C05505=1108.942,119.637,-59.989,-179.645,8.357,149.505
C05506=1108.947,119.424,-59.972,-179.646,8.354,149.505
C05507=1108.951,119.210,-59.955,-179.648,8.352,149.505
C05508=1108.955,118.996,-59.937,-179.649,8.349,149.504
C05509=1108.959,118.783,-59.919,-179.651,8.345,149.504
C05510=1108.963,118.569,-59.902,-179.652,8.342,149.504
C05511=1108.967,118.356,-59.885,-179.653,8.340,149.504
C05512=1108.971,118.142,-59.867,-179.655,8.337,149.503
C05513=1108.975,117.929,-59.849,-179.656,8.334,149.503
C05514=1108.979,117.680,-59.829,-179.658,8.331,149.503
C05515=1108.985,117.430,-59.809,-179.660,8.327,149.503
C05516=1108.989,117.181,-59.788,-179.661,8.324,149.502
C05517=1108.994,116.932,-59.768,-179.664,8.321,149.502
C05518=1108.998,116.683,-59.748,-179.666,8.317,149.502
C05519=1109.004,116.433,-59.727,-179.667,8.313,149.501
C05520=1109.008,116.184,-59.707,-179.669,8.310,149.501
C05521=1109.013,115.935,-59.687,-179.671,8.307,149.501
C05522=1109.017,115.686,-59.666,-179.672,8.303,149.500
C05523=1109.023,115.436,-59.646,-179.674,8.300,149.500
C05524=1109.027,115.187,-59.626,-179.676,8.297,149.500
C05525=1109.031,114.938,-59.605,-179.677,8.293,149.499
C05526=1109.036,114.689,-59.586,-179.679,8.290,149.499
C05527=1109.041,114.441,-59.566,-179.681,8.287,149.499
C05528=1109.046,114.191,-59.545,-179.683,8.283,149.499
C05529=1109.051,113.942,-59.525,-179.685,8.279,149.498
C05530=1109.056,113.693,-59.505,-179.686,8.277,149.498
C05531=1109.060,113.444,-59.484,-179.688,8.273,149.498
C05532=1109.065,113.194,-59.464,-179.690,8.269,149.497
C05533=1109.069,112.945,-59.444,-179.692,8.266,149.497
C05534=1109.074,112.696,-59.423,-179.693,8.263,149.497
C05535=1109.080,112.447,-59.404,-179.695,8.259,149.497
C05536=1109.084,112.198,-59.383,-179.697,8.256,149.496
C05537=1109.089,111.949,-59.364,-179.698,8.253,149.496
C05538=1109.093,111.700,-59.343,-179.700,8.249,149.496
C05539=1109.098,111.450,-59.324,-179.702,8.246,149.495
C05540=1109.102,111.201,-59.303,-179.704,8.242,149.495
C05541=1109.108,110.952,-59.284,-179.706,8.238,149.495
C05542=1109.112,110.703,-59.264,-179.708,8.235,149.495
C05543=1109.117,110.454,-59.244,-179.709,8.231,149.494
C05544=1109.122,110.205,-59.223,-179.711,8.227,149.494
C05545=1109.127,109.955,-59.203,-179.713,8.224,149.494
C05546=1109.131,109.706,-59.183,-179.715,8.220,149.493
C05547=1109.137,109.457,-59.164,-179.717,8.216,149.493
C05548=1109.141,109.208,-59.143,-179.719,8.213,149.493
C05549=1109.146,108.959,-59.124,-179.721,8.209,149.493
C05550=1109.150,108.710,-59.103,-179.723,8.206,149.492
C05551=1109.156,108.461,-59.084,-179.725,8.202,149.492
C05552=1109.160,108.211,-59.064,-179.726,8.198,149.491
C05553=1109.165,107.962,-59.044,-179.729,8.195,149.491
C05554=1109.170,107.713,-59.024,-179.731,8.191,149.491
C05555=1109.174,107.463,-59.005,-179.732,8.187,149.491
C05556=1109.179,107.215,-58.985,-179.734,8.185,149.490
C05557=1109.184,106.965,-58.965,-179.735,8.181,149.490
C05558=1109.188,106.716,-58.946,-179.737,8.177,149.490
C05559=1109.193,106.467,-58.926,-179.739,8.173,149.489
C05560=1109.198,106.218,-58.906,-179.741,8.170,149.489
C05561=1109.203,105.969,-58.887,-179.743,8.166,149.489
C05562=1109.207,105.755,-58.869,-179.745,8.162,149.488
C05563=1109.210,105.542,-58.853,-179.746,8.159,149.488
C05564=1109.215,105.328,-58.835,-179.748,8.156,149.488
C05565=1109.219,105.114,-58.819,-179.749,8.153,149.488
C05566=1109.223,104.901,-58.802,-179.750,8.150,149.487
C05567=1109.227,104.687,-58.785,-179.752,8.146,149.487
C05568=1109.231,104.473,-58.768,-179.754,8.144,149.487
C05569=1109.235,104.259,-58.752,-179.755,8.141,149.486
C05570=1109.240,104.010,-58.732,-179.757,8.137,149.486
C05571=1109.245,103.761,-58.713,-179.758,8.133,149.486
C05572=1109.249,103.512,-58.692,-179.760,8.129,149.485
C05573=1109.255,103.263,-58.673,-179.762,8.126,149.485
C05574=1109.260,103.013,-58.653,-179.763,8.122,149.484
C05575=1109.264,102.764,-58.634,-179.765,8.118,149.484
C05576=1109.269,102.515,-58.615,-179.767,8.114,149.484
C05577=1109.274,102.266,-58.595,-179.769,8.111,149.483
C05578=1109.278,102.016,-58.576,-179.770,8.107,149.483
C05579=1109.284,101.767,-58.556,-179.772,8.103,149.482
C05580=1109.288,101.518,-58.537,-179.774,8.099,149.482
C05581=1109.292,101.269,-58.517,-179.776,8.096,149.482
C05582=1109.297,101.020,-58.498,-179.777,8.092,149.481
C05583=1109.302,100.771,-58.478,-179.778,8.089,149.481
C05584=1109.307,100.522,-58.459,-179.780,8.085,149.481
C05585=1109.312,100.273,-58.440,-179.781,8.081,149.480
C05586=1109.316,100.023,-58.420,-179.783,8.077,149.480
C05587=1109.322,99.774,-58.401,-179.785,8.073,149.479
C05588=1109.326,99.525,-58.382,-179.787,8.069,149.479
C05589=1109.331,99.276,-58.362,-179.788,8.066,149.479
C05590=1109.336,99.026,-58.343,-179.790,8.062,149.478
C05591=1109.340,98.777,-58.324,-179.791,8.058,149.478
C05592=1109.345,98.528,-58.304,-179.792,8.055,149.477
C05593=1109.350,98.278,-58.285,-179.794,8.051,149.477
C05594=1109.356,98.029,-58.266,-179.796,8.047,149.476
C05595=1109.360,97.780,-58.247,-179.797,8.043,149.476
C05596=1109.365,97.531,-58.228,-179.799,8.039,149.475
C05597=1109.369,97.282,-58.209,-179.800,8.035,149.475
C05598=1109.374,97.032,-58.189,-179.802,8.031,149.475
C05599=1109.379,96.783,-58.170,-179.803,8.028,149.474
C05600=1109.383,96.534,-58.151,-179.805,8.024,149.474
C05601=1109.388,96.285,-58.131,-179.806,8.021,149.473
C05602=1109.393,96.035,-58.113,-179.808,8.017,149.473
C05603=1109.398,95.787,-58.094,-179.809,8.013,149.472
C05604=1109.403,95.537,-58.074,-179.811,8.009,149.472
C05605=1109.407,95.288,-58.055,-179.812,8.006,149.472
C05606=1109.412,95.039,-58.036,-179.814,8.002,149.471
C05607=1109.418,94.789,-58.017,-179.815,7.998,149.471
C05608=1109.422,94.540,-57.998,-179.816,7.994,149.470
C05609=1109.427,94.291,-57.979,-179.818,7.990,149.470
C05610=1109.431,94.042,-57.960,-179.819,7.987,149.469
C05611=1109.437,93.792,-57.941,-179.820,7.983,149.469
C05612=1109.441,93.543,-57.922,-179.822,7.979,149.468
C05613=1109.446,93.294,-57.903,-179.824,7.975,149.468
C05614=1109.450,93.045,-57.884,-179.825,7.971,149.467
C05615=1109.456,92.796,-57.865,-179.826,7.968,149.467
C05616=1109.460,92.546,-57.846,-179.827,7.964,149.466
C05617=1109.465,92.297,-57.827,-179.829,7.960,149.466
C05618=1109.469,92.083,-57.811,-179.830,7.957,149.466
C05619=1109.473,91.870,-57.795,-179.831,7.954,149.465
C05620=1109.478,91.656,-57.778,-179.833,7.950,149.465
C05621=1109.482,91.441,-57.762,-179.833,7.947,149.464
C05622=1109.486,91.228,-57.747,-179.834,7.944,149.464
C05623=1109.490,91.015,-57.730,-179.836,7.941,149.464
C05624=1109.493,90.801,-57.714,-179.837,7.937,149.463
C05625=1109.498,90.587,-57.698,-179.838,7.934,149.463
C05626=1109.503,90.338,-57.678,-179.840,7.930,149.462
C05627=1109.507,90.088,-57.660,-179.841,7.926,149.462
C05628=1109.513,89.840,-57.641,-179.842,7.923,149.461
C05629=1109.517,89.590,-57.623,-179.844,7.919,149.461
C05630=1109.522,89.341,-57.603,-179.844,7.915,149.460
C05631=1109.527,89.091,-57.585,-179.846,7.911,149.460
C05632=1109.531,88.842,-57.566,-179.847,7.907,149.459
C05633=1109.537,88.593,-57.548,-179.849,7.903,149.459
C05634=1109.541,88.344,-57.529,-179.850,7.900,149.458
C05635=1109.547,88.094,-57.510,-179.851,7.896,149.458
C05636=1109.551,87.845,-57.491,-179.852,7.892,149.457
C05637=1109.556,87.596,-57.473,-179.853,7.889,149.457
C05638=1109.561,87.347,-57.454,-179.854,7.884,149.456
C05639=1109.565,87.097,-57.435,-179.856,7.881,149.456
C05640=1109.570,86.848,-57.417,-179.857,7.877,149.455
C05641=1109.576,86.599,-57.398,-179.858,7.873,149.454
C05642=1109.580,86.350,-57.379,-179.860,7.869,149.454
C05643=1109.584,86.100,-57.361,-179.861,7.866,149.454
C05644=1109.590,85.851,-57.343,-179.862,7.862,149.453
C05645=1109.594,85.602,-57.323,-179.863,7.858,149.453
C05646=1109.599,85.353,-57.305,-179.864,7.854,149.452
C05647=1109.604,85.104,-57.286,-179.865,7.851,149.451
C05648=1109.609,84.854,-57.268,-179.867,7.846,149.451
C05649=1109.614,84.605,-57.250,-179.868,7.843,149.450
C05650=1109.619,84.356,-57.231,-179.869,7.839,149.450
C05651=1109.623,84.106,-57.212,-179.870,7.836,149.449
C05652=1109.628,83.857,-57.194,-179.871,7.832,149.449
C05653=1109.633,83.608,-57.176,-179.872,7.828,149.448
C05654=1109.638,83.358,-57.157,-179.873,7.825,149.448
C05655=1109.643,83.109,-57.139,-179.874,7.820,149.447
C05656=1109.647,82.860,-57.120,-179.875,7.817,149.447
C05657=1109.652,82.611,-57.102,-179.877,7.813,149.446
C05658=1109.657,82.361,-57.083,-179.878,7.809,149.446
C05659=1109.662,82.112,-57.065,-179.879,7.805,149.445
C05660=1109.667,81.863,-57.046,-179.880,7.802,149.445
C05661=1109.671,81.613,-57.028,-179.881,7.798,149.444
C05662=1109.676,81.364,-57.010,-179.882,7.794,149.443
C05663=1109.682,81.115,-56.991,-179.883,7.791,149.443
C05664=1109.686,80.866,-56.973,-179.884,7.787,149.442
C05665=1109.691,80.616,-56.954,-179.885,7.783,149.442
C05666=1109.696,80.367,-56.936,-179.887,7.779,149.441
C05667=1109.700,80.118,-56.918,-179.887,7.776,149.441
C05668=1109.706,79.868,-56.900,-179.889,7.772,149.440
C05669=1109.710,79.618,-56.882,-179.889,7.769,149.440
C05670=1109.715,79.370,-56.863,-179.891,7.765,149.439
C05671=1109.720,79.121,-56.845,-179.891,7.761,149.438
C05672=1109.725,78.872,-56.827,-179.892,7.757,149.438
C05673=1109.730,78.622,-56.809,-179.893,7.754,149.437
C05674=1109.734,78.408,-56.793,-179.894,7.751,149.437
C05675=1109.738,78.194,-56.778,-179.895,7.747,149.436
C05676=1109.742,77.980,-56.762,-179.896,7.744,149.436
C05677=1109.747,77.767,-56.746,-179.897,7.741,149.435
C05678=1109.751,77.552,-56.731,-179.898,7.738,149.435
C05679=1109.755,77.339,-56.715,-179.899,7.735,149.435
C05680=1109.759,77.125,-56.699,-179.899,7.731,149.434
C05681=1109.763,76.911,-56.684,-179.900,7.728,149.433
C05682=1109.768,76.662,-56.666,-179.902,7.724,149.433
C05683=1109.773,76.413,-56.647,-179.903,7.720,149.433
C05684=1109.777,76.163,-56.629,-179.904,7.716,149.432
C05685=1109.782,75.914,-56.611,-179.906,7.712,149.432
C05686=1109.787,75.665,-56.593,-179.907,7.708,149.431
C05687=1109.792,75.415,-56.575,-179.909,7.704,149.431
C05688=1109.797,75.166,-56.557,-179.910,7.700,149.430
C05689=1109.802,74.917,-56.539,-179.912,7.696,149.430
C05690=1109.806,74.667,-56.520,-179.913,7.693,149.429
C05691=1109.811,74.418,-56.502,-179.914,7.689,149.428
C05692=1109.816,74.168,-56.485,-179.915,7.685,149.428
C05693=1109.821,73.919,-56.467,-179.917,7.681,149.428
C05694=1109.826,73.670,-56.449,-179.919,7.677,149.427
C05695=1109.831,73.421,-56.431,-179.920,7.673,149.427
C05696=1109.836,73.172,-56.413,-179.921,7.669,149.426
C05697=1109.841,72.922,-56.395,-179.923,7.665,149.426
C05698=1109.845,72.672,-56.377,-179.924,7.661,149.425
C05699=1109.850,72.423,-56.359,-179.926,7.657,149.425
C05700=1109.855,72.174,-56.341,-179.926,7.654,149.424
C05701=1109.860,71.924,-56.324,-179.928,7.649,149.423
C05702=1109.865,71.675,-56.306,-179.929,7.645,149.423
C05703=1109.869,71.426,-56.288,-179.931,7.642,149.423
C05704=1109.874,71.177,-56.270,-179.932,7.637,149.422
C05705=1109.879,70.928,-56.252,-179.933,7.633,149.422
C05706=1109.884,70.679,-56.234,-179.935,7.629,149.421
C05707=1109.889,70.429,-56.217,-179.936,7.625,149.420
C05708=1109.894,70.180,-56.199,-179.938,7.621,149.420
C05709=1109.899,69.931,-56.181,-179.939,7.618,149.420
C05710=1109.904,69.681,-56.163,-179.940,7.614,149.419
C05711=1109.909,69.432,-56.146,-179.941,7.610,149.418
C05712=1109.913,69.182,-56.128,-179.943,7.606,149.418
C05713=1109.918,68.933,-56.110,-179.944,7.602,149.417
C05714=1109.923,68.684,-56.092,-179.946,7.598,149.417
C05715=1109.928,68.434,-56.075,-179.947,7.594,149.417
C05716=1109.933,68.185,-56.057,-179.948,7.590,149.416
C05717=1109.938,67.936,-56.039,-179.950,7.586,149.415
C05718=1109.942,67.686,-56.022,-179.951,7.583,149.415
C05719=1109.947,67.437,-56.004,-179.952,7.578,149.414
C05720=1109.952,67.188,-55.986,-179.953,7.574,149.414
C05721=1109.957,66.938,-55.969,-179.955,7.571,149.414
C05722=1109.962,66.689,-55.951,-179.956,7.566,149.413
C05723=1109.967,66.439,-55.934,-179.958,7.562,149.412
C05724=1109.972,66.190,-55.916,-179.959,7.558,149.412
C05725=1109.977,65.941,-55.899,-179.960,7.555,149.411
C05726=1109.982,65.691,-55.881,-179.961,7.551,149.411
C05727=1109.986,65.442,-55.864,-179.962,7.547,149.410
C05728=1109.991,65.192,-55.847,-179.964,7.543,149.410
C05729=1109.997,64.944,-55.829,-179.966,7.539,149.409
C05730=1110.000,64.730,-55.814,-179.966,7.535,149.409
C05731=1110.005,64.516,-55.799,-179.968,7.532,149.408
C05732=1110.009,64.302,-55.784,-179.969,7.528,149.408
C05733=1110.013,64.088,-55.769,-179.970,7.525,149.407
C05734=1110.017,63.874,-55.754,-179.970,7.522,149.407
C05735=1110.021,63.660,-55.739,-179.972,7.518,149.407
C05736=1110.026,63.446,-55.724,-179.973,7.515,149.406
C05737=1110.029,63.232,-55.709,-179.974,7.512,149.406
C05738=1110.034,62.982,-55.691,-179.975,7.508,149.405
C05739=1110.040,62.733,-55.674,-179.977,7.504,149.405
C05740=1110.044,62.485,-55.657,-179.978,7.500,149.404
C05741=1110.050,62.235,-55.640,-179.979,7.496,149.404
C05742=1110.055,61.985,-55.623,-179.981,7.492,149.403
C05743=1110.059,61.736,-55.605,-179.981,7.488,149.402
C05744=1110.064,61.486,-55.588,-179.983,7.484,149.402
C05745=1110.068,61.237,-55.571,-179.984,7.480,149.401
C05746=1110.074,60.988,-55.553,-179.986,7.476,149.401
C05747=1110.079,60.738,-55.536,-179.987,7.472,149.400
C05748=1110.083,60.489,-55.519,-179.988,7.468,149.400
C05749=1110.089,60.240,-55.502,-179.989,7.465,149.399
C05750=1110.094,59.990,-55.484,-179.990,7.460,149.399
C05751=1110.098,59.741,-55.467,-179.992,7.457,149.398
C05752=1110.103,59.491,-55.450,-179.993,7.452,149.398
C05753=1110.108,59.242,-55.433,-179.994,7.448,149.397
C05754=1110.113,58.993,-55.415,-179.996,7.444,149.397
C05755=1110.117,58.743,-55.399,-179.996,7.441,149.396
C05756=1110.123,58.494,-55.382,-179.998,7.437,149.396
C05757=1110.127,58.245,-55.364,-179.999,7.433,149.395
C05758=1110.132,57.995,-55.347,180.000,7.428,149.394
C05759=1110.138,57.746,-55.330,179.998,7.425,149.394
C05760=1110.142,57.496,-55.313,179.997,7.420,149.393
C05761=1110.148,57.248,-55.295,179.996,7.417,149.393
C05762=1110.152,56.998,-55.279,179.995,7.413,149.392
C05763=1110.157,56.748,-55.262,179.994,7.409,149.392
C05764=1110.162,56.499,-55.245,179.992,7.405,149.391
C05765=1110.167,56.249,-55.228,179.991,7.401,149.391
C05766=1110.172,56.001,-55.211,179.990,7.397,149.390
C05767=1110.177,55.751,-55.193,179.989,7.393,149.389
C05768=1110.182,55.502,-55.177,179.988,7.389,149.389
C05769=1110.186,55.252,-55.160,179.987,7.385,149.388
C05770=1110.192,55.003,-55.143,179.985,7.381,149.388
C05771=1110.196,54.754,-55.126,179.984,7.377,149.387
C05772=1110.202,54.504,-55.109,179.983,7.373,149.387
C05773=1110.206,54.254,-55.092,179.982,7.369,149.386
C05774=1110.211,54.006,-55.075,179.981,7.365,149.386
C05775=1110.216,53.756,-55.058,179.979,7.361,149.385
C05776=1110.221,53.507,-55.041,179.978,7.357,149.384
C05777=1110.226,53.257,-55.024,179.977,7.353,149.384
C05778=1110.231,53.008,-55.008,179.976,7.349,149.383
C05779=1110.236,52.759,-54.991,179.975,7.345,149.383
C05780=1110.240,52.509,-54.974,179.974,7.341,149.382
C05781=1110.245,52.260,-54.957,179.972,7.337,149.382
C05782=1110.251,52.011,-54.940,179.972,7.334,149.381
C05783=1110.255,51.761,-54.924,179.970,7.329,149.381
C05784=1110.260,51.511,-54.906,179.969,7.325,149.380
C05785=1110.266,51.262,-54.890,179.968,7.321,149.379
C05786=1110.270,51.049,-54.876,179.967,7.318,149.379
C05787=1110.273,50.834,-54.862,179.966,7.314,149.378
C05788=1110.278,50.620,-54.847,179.965,7.310,149.378
C05789=1110.282,50.405,-54.833,179.964,7.307,149.377
C05790=1110.286,50.192,-54.819,179.963,7.304,149.377
C05791=1110.290,49.978,-54.804,179.963,7.301,149.376
C05792=1110.295,49.763,-54.790,179.961,7.297,149.376
C05793=1110.299,49.550,-54.775,179.960,7.294,149.376
C05794=1110.304,49.300,-54.759,179.959,7.289,149.375
C05795=1110.309,49.051,-54.742,179.958,7.285,149.374
C05796=1110.314,48.802,-54.725,179.957,7.282,149.374
C05797=1110.318,48.552,-54.708,179.956,7.278,149.373
C05798=1110.324,48.303,-54.693,179.955,7.273,149.372
C05799=1110.328,48.053,-54.676,179.954,7.269,149.372
C05800=1110.334,47.803,-54.659,179.952,7.265,149.371
C05801=1110.339,47.555,-54.643,179.952,7.262,149.371
C05802=1110.343,47.305,-54.626,179.951,7.257,149.370
C05803=1110.348,47.056,-54.609,179.949,7.253,149.370
C05804=1110.354,46.806,-54.593,179.948,7.249,149.369
C05805=1110.358,46.556,-54.576,179.947,7.245,149.368
C05806=1110.363,46.308,-54.560,179.946,7.241,149.368
C05807=1110.368,46.058,-54.543,179.945,7.237,149.367
C05808=1110.373,45.808,-54.528,179.944,7.233,149.367
C05809=1110.378,45.559,-54.511,179.943,7.229,149.366
C05810=1110.383,45.310,-54.494,179.942,7.225,149.365
C05811=1110.388,45.061,-54.478,179.941,7.221,149.365
C05812=1110.393,44.811,-54.462,179.940,7.217,149.364
C05813=1110.398,44.562,-54.445,179.939,7.213,149.364
C05814=1110.402,44.312,-54.429,179.937,7.208,149.363
C05815=1110.407,44.063,-54.412,179.937,7.205,149.362
C05816=1110.413,43.813,-54.396,179.935,7.201,149.362
C05817=1110.417,43.564,-54.379,179.934,7.197,149.361
C05818=1110.422,43.315,-54.363,179.933,7.192,149.361
C05819=1110.427,43.065,-54.347,179.932,7.188,149.360
C05820=1110.432,42.816,-54.331,179.932,7.185,149.359
C05821=1110.437,42.566,-54.315,179.930,7.181,149.359
C05822=1110.442,42.317,-54.298,179.929,7.176,149.358
C05823=1110.447,42.068,-54.282,179.928,7.172,149.357
C05824=1110.451,41.818,-54.266,179.928,7.169,149.357
C05825=1110.457,41.568,-54.249,179.927,7.164,149.356
C05826=1110.462,41.318,-54.233,179.925,7.160,149.356
C05827=1110.467,41.070,-54.217,179.924,7.156,149.355
C05828=1110.472,40.820,-54.200,179.923,7.152,149.354
C05829=1110.477,40.571,-54.184,179.922,7.148,149.354
C05830=1110.481,40.321,-54.168,179.921,7.144,149.353
C05831=1110.487,40.072,-54.152,179.920,7.140,149.352
C05832=1110.491,39.822,-54.135,179.919,7.135,149.352
C05833=1110.497,39.573,-54.120,179.918,7.131,149.351
C05834=1110.502,39.324,-54.104,179.918,7.127,149.351
C05835=1110.507,39.074,-54.088,179.917,7.123,149.350
C05836=1110.512,38.825,-54.071,179.916,7.119,149.349
C05837=1110.516,38.575,-54.055,179.914,7.115,149.349
C05838=1110.522,38.326,-54.039,179.914,7.111,149.348
C05839=1110.526,38.076,-54.023,179.912,7.107,149.347
C05840=1110.531,37.827,-54.007,179.911,7.103,149.347
C05841=1110.536,37.577,-53.991,179.910,7.099,149.346
C05842=1110.541,37.363,-53.977,179.910,7.095,149.345
C05843=1110.545,37.149,-53.964,179.909,7.092,149.345
C05844=1110.550,36.935,-53.950,179.908,7.088,149.344
C05845=1110.554,36.721,-53.936,179.907,7.084,149.344
C05846=1110.558,36.507,-53.922,179.907,7.081,149.343
C05847=1110.562,36.293,-53.908,179.906,7.077,149.343
C05848=1110.566,36.079,-53.895,179.905,7.073,149.342
C05849=1110.570,35.864,-53.881,179.904,7.070,149.342
C05850=1110.576,35.615,-53.866,179.903,7.066,149.341
C05851=1110.580,35.366,-53.849,179.903,7.062,149.340
C05852=1110.585,35.116,-53.834,179.902,7.058,149.340
C05853=1110.591,34.867,-53.818,179.900,7.054,149.339
C05854=1110.595,34.617,-53.801,179.899,7.049,149.338
C05855=1110.601,34.368,-53.786,179.899,7.046,149.338
C05856=1110.605,34.118,-53.770,179.898,7.041,149.337
C05857=1110.610,33.869,-53.753,179.897,7.037,149.336
C05858=1110.615,33.620,-53.738,179.896,7.033,149.336
C05859=1110.620,33.370,-53.723,179.895,7.028,149.335
C05860=1110.625,33.120,-53.707,179.894,7.025,149.334
C05861=1110.630,32.872,-53.691,179.893,7.021,149.334
C05862=1110.635,32.621,-53.675,179.892,7.016,149.333
C05863=1110.641,32.372,-53.659,179.891,7.012,149.332
C05864=1110.645,32.122,-53.644,179.890,7.007,149.332
C05865=1110.650,31.873,-53.627,179.890,7.004,149.331
C05866=1110.655,31.624,-53.612,179.889,6.999,149.330
C05867=1110.660,31.374,-53.596,179.888,6.995,149.330
C05868=1110.665,31.125,-53.580,179.887,6.991,149.329
C05869=1110.670,30.875,-53.565,179.886,6.987,149.328
C05870=1110.674,30.626,-53.549,179.885,6.983,149.328
C05871=1110.680,30.377,-53.533,179.884,6.979,149.327
C05872=1110.685,30.127,-53.517,179.884,6.974,149.326
C05873=1110.690,29.878,-53.502,179.883,6.970,149.325
C05874=1110.695,29.628,-53.487,179.882,6.966,149.325
C05875=1110.700,29.379,-53.471,179.881,6.962,149.324
C05876=1110.705,29.129,-53.455,179.880,6.958,149.323
C05877=1110.709,28.879,-53.440,179.880,6.953,149.323
C05878=1110.715,28.630,-53.424,179.878,6.949,149.322
C05879=1110.720,28.381,-53.408,179.878,6.945,149.321
C05880=1110.725,28.132,-53.393,179.877,6.941,149.321
C05881=1110.729,27.882,-53.377,179.876,6.936,149.320
C05882=1110.735,27.633,-53.362,179.875,6.932,149.319
C05883=1110.740,27.383,-53.346,179.875,6.928,149.318
C05884=1110.744,27.133,-53.331,179.874,6.924,149.318
C05885=1110.750,26.884,-53.315,179.873,6.920,149.317
C05886=1110.755,26.635,-53.299,179.872,6.915,149.316
C05887=1110.760,26.386,-53.284,179.871,6.911,149.316
C05888=1110.764,26.135,-53.268,179.871,6.907,149.315
C05889=1110.770,25.886,-53.253,179.870,6.902,149.314
C05890=1110.774,25.637,-53.238,179.869,6.898,149.313
C05891=1110.780,25.388,-53.222,179.868,6.894,149.313
C05892=1110.785,25.138,-53.207,179.867,6.889,149.312
C05893=1110.789,24.888,-53.191,179.867,6.886,149.311
C05894=1110.795,24.639,-53.176,179.866,6.881,149.311
C05895=1110.800,24.389,-53.162,179.865,6.877,149.310
C05896=1110.805,24.140,-53.146,179.864,6.872,149.309
C05897=1110.810,23.890,-53.130,179.863,6.868,149.308
C05898=1110.814,23.676,-53.117,179.863,6.864,149.308
C05899=1110.818,23.462,-53.104,179.862,6.861,149.307
C05900=1110.823,23.247,-53.091,179.862,6.857,149.306
C05901=1110.827,23.034,-53.078,179.861,6.853,149.306
C05902=1110.831,22.819,-53.064,179.861,6.849,149.305
C05903=1110.836,22.605,-53.051,179.860,6.846,149.304
C05904=1110.839,22.391,-53.038,179.860,6.842,149.304
C05905=1110.845,22.176,-53.025,179.858,6.838,149.303
C05906=1110.849,21.926,-53.010,179.858,6.835,149.302
C05907=1110.854,21.677,-52.994,179.857,6.830,149.302
C05908=1110.859,21.428,-52.979,179.857,6.826,149.301
C05909=1110.864,21.179,-52.964,179.856,6.821,149.300
C05910=1110.869,20.930,-52.949,179.855,6.817,149.299
C05911=1110.874,20.679,-52.934,179.855,6.813,149.299
C05912=1110.879,20.430,-52.919,179.854,6.808,149.298
C05913=1110.884,20.180,-52.903,179.853,6.804,149.297
C05914=1110.888,19.931,-52.888,179.852,6.799,149.296
C05915=1110.894,19.681,-52.873,179.851,6.795,149.296
C05916=1110.899,19.432,-52.858,179.851,6.791,149.295
C05917=1110.904,19.183,-52.843,179.850,6.787,149.294
C05918=1110.909,18.934,-52.828,179.850,6.782,149.293
C05919=1110.915,18.684,-52.813,179.849,6.778,149.293
C05920=1110.919,18.434,-52.798,179.848,6.773,149.292
C05921=1110.924,18.184,-52.782,179.848,6.769,149.291
C05922=1110.929,17.935,-52.767,179.847,6.765,149.290
C05923=1110.934,17.685,-52.752,179.846,6.760,149.289
C05924=1110.939,17.436,-52.737,179.846,6.756,149.289
C05925=1110.944,17.186,-52.723,179.845,6.751,149.288
C05926=1110.949,16.937,-52.707,179.844,6.747,149.287
C05927=1110.954,16.688,-52.692,179.844,6.743,149.286
C05928=1110.960,16.438,-52.677,179.843,6.739,149.285
C05929=1110.964,16.189,-52.662,179.842,6.734,149.285
C05930=1110.969,15.939,-52.648,179.842,6.729,149.284
C05931=1110.975,15.690,-52.632,179.841,6.725,149.283
C05932=1110.979,15.441,-52.617,179.841,6.721,149.282
C05933=1110.985,15.191,-52.602,179.840,6.716,149.281
C05934=1110.989,14.941,-52.587,179.839,6.712,149.281
C05935=1110.994,14.691,-52.573,179.839,6.707,149.280
C05936=1110.999,14.442,-52.557,179.838,6.702,149.279
C05937=1111.004,14.192,-52.543,179.837,6.698,149.278
C05938=1111.009,13.943,-52.528,179.837,6.694,149.277
C05939=1111.015,13.693,-52.513,179.837,6.689,149.276
C05940=1111.019,13.444,-52.498,179.836,6.685,149.276
C05941=1111.024,13.194,-52.484,179.835,6.680,149.275
C05942=1111.030,12.945,-52.468,179.834,6.676,149.274
C05943=1111.035,12.695,-52.454,179.834,6.671,149.273
C05944=1111.039,12.446,-52.439,179.833,6.668,149.272
C05945=1111.044,12.196,-52.425,179.833,6.663,149.272
C05946=1111.050,11.947,-52.409,179.832,6.658,149.271
C05947=1111.055,11.697,-52.395,179.832,6.653,149.270
C05948=1111.059,11.448,-52.380,179.831,6.649,149.269
C05949=1111.065,11.198,-52.365,179.830,6.644,149.268
C05950=1111.070,10.949,-52.350,179.830,6.640,149.267
C05951=1111.075,10.699,-52.336,179.830,6.636,149.266
C05952=1111.079,10.449,-52.321,179.829,6.631,149.266
C05953=1111.085,10.200,-52.306,179.829,6.626,149.265
C05954=1111.089,9.986,-52.294,179.828,6.623,149.264
C05955=1111.093,9.771,-52.281,179.827,6.618,149.263
C05956=1111.098,9.557,-52.269,179.827,6.615,149.263
C05957=1111.102,9.343,-52.256,179.827,6.611,149.262
C05958=1111.106,9.129,-52.244,179.826,6.607,149.261
C05959=1111.111,8.914,-52.231,179.826,6.603,149.260
C05960=1111.115,8.700,-52.218,179.826,6.599,149.260
C05961=1111.119,8.486,-52.206,179.825,6.596,149.259
C05962=1111.125,8.236,-52.191,179.825,6.591,149.258
C05963=1111.130,7.987,-52.176,179.824,6.586,149.257
C05964=1111.135,7.737,-52.162,179.823,6.582,149.256
C05965=1111.140,7.487,-52.148,179.823,6.577,149.255
C05966=1111.144,7.238,-52.133,179.822,6.573,149.255
C05967=1111.149,6.988,-52.118,179.821,6.568,149.254
C05968=1111.155,6.738,-52.104,179.821,6.563,149.253
C05969=1111.160,6.489,-52.090,179.820,6.558,149.252
C05970=1111.165,6.240,-52.075,179.820,6.554,149.251
C05971=1111.170,5.991,-52.060,179.819,6.549,149.250
C05972=1111.175,5.741,-52.046,179.818,6.545,149.250
C05973=1111.180,5.491,-52.032,179.818,6.540,149.249
C05974=1111.185,5.241,-52.018,179.817,6.535,149.248
C05975=1111.190,4.992,-52.003,179.817,6.531,149.247
C05976=1111.195,4.743,-51.988,179.816,6.526,149.246
C05977=1111.201,4.493,-51.974,179.816,6.522,149.245
C05978=1111.206,4.244,-51.960,179.815,6.518,149.245
C05979=1111.211,3.994,-51.945,179.815,6.513,149.244
C05980=1111.216,3.744,-51.931,179.814,6.509,149.243
C05981=1111.220,3.495,-51.916,179.813,6.504,149.242
C05982=1111.225,3.245,-51.902,179.812,6.499,149.241
C05983=1111.230,2.996,-51.887,179.812,6.494,149.240
C05984=1111.236,2.747,-51.874,179.811,6.490,149.240
C05985=1111.241,2.497,-51.859,179.810,6.485,149.239
C05986=1111.246,2.247,-51.845,179.810,6.481,149.238
C05987=1111.251,1.998,-51.831,179.809,6.476,149.237
C05988=1111.256,1.748,-51.816,179.808,6.472,149.236
C05989=1111.261,1.499,-51.803,179.808,6.468,149.235
C05990=1111.266,1.249,-51.788,179.808,6.463,149.235
C05991=1111.271,0.999,-51.774,179.807,6.458,149.234
C05992=1111.276,0.750,-51.760,179.806,6.454,149.233
C05993=1111.281,0.501,-51.745,179.806,6.449,149.232
C05994=1111.286,0.252,-51.731,179.805,6.445,149.231
C05995=1111.291,0.002,-51.717,179.805,6.440,149.230
C05996=1111.296,-0.248,-51.702,179.804,6.435,149.230
C05997=1111.301,-0.498,-51.688,179.803,6.431,149.229
C05998=1111.306,-0.748,-51.674,179.803,6.426,149.228
C05999=1111.312,-0.997,-51.660,179.802,6.422,149.227
C06000=1111.317,-1.247,-51.646,179.802,6.418,149.226
C06001=1111.322,-1.496,-51.632,179.801,6.413,149.225
C06002=1111.327,-1.746,-51.618,179.801,6.408,149.225
C06003=1111.332,-1.995,-51.604,179.800,6.404,149.224
C06004=1111.337,-2.244,-51.590,179.799,6.399,149.223
C06005=1111.341,-2.494,-51.576,179.799,6.395,149.222
C06006=1111.346,-2.744,-51.561,179.798,6.390,149.221
C06007=1111.352,-2.993,-51.548,179.797,6.386,149.221
C06008=1111.357,-3.243,-51.533,179.797,6.381,149.220
C06009=1111.362,-3.492,-51.519,179.796,6.376,149.219
C06010=1111.367,-3.707,-51.508,179.796,6.373,149.218
C06011=1111.371,-3.921,-51.495,179.795,6.369,149.217
C06012=1111.375,-4.135,-51.483,179.794,6.365,149.217
C06013=1111.380,-4.350,-51.472,179.794,6.361,149.216
C06014=1111.384,-4.565,-51.460,179.794,6.358,149.215
C06015=1111.388,-4.778,-51.448,179.793,6.353,149.215
C06016=1111.392,-4.994,-51.436,179.793,6.349,149.214
C06017=1111.397,-5.208,-51.424,179.792,6.346,149.213
C06018=1111.402,-5.457,-51.410,179.792,6.341,149.212
C06019=1111.407,-5.706,-51.396,179.791,6.337,149.212
C06020=1111.413,-5.957,-51.382,179.790,6.332,149.211
C06021=1111.417,-6.206,-51.368,179.790,6.327,149.210
C06022=1111.422,-6.455,-51.354,179.789,6.323,149.209
C06023=1111.427,-6.705,-51.340,179.788,6.318,149.208
C06024=1111.433,-6.955,-51.327,179.788,6.314,149.207
C06025=1111.438,-7.204,-51.313,179.788,6.310,149.207
C06026=1111.442,-7.454,-51.299,179.787,6.305,149.206
C06027=1111.447,-7.703,-51.285,179.786,6.301,149.205
C06028=1111.453,-7.953,-51.272,179.786,6.296,149.204
C06029=1111.458,-8.203,-51.257,179.785,6.291,149.203
C06030=1111.463,-8.451,-51.244,179.784,6.287,149.203
C06031=1111.468,-8.702,-51.230,179.784,6.282,149.202
C06032=1111.473,-8.951,-51.216,179.783,6.277,149.201
C06033=1111.479,-9.200,-51.202,179.783,6.273,149.200
C06034=1111.483,-9.450,-51.189,179.782,6.269,149.199
C06035=1111.488,-9.700,-51.175,179.782,6.264,149.198
C06036=1111.494,-9.949,-51.161,179.781,6.260,149.197
C06037=1111.498,-10.199,-51.148,179.780,6.255,149.197
C06038=1111.504,-10.448,-51.134,179.780,6.251,149.196
C06039=1111.509,-10.698,-51.121,179.779,6.246,149.195
C06040=1111.513,-10.948,-51.107,179.779,6.241,149.194
C06041=1111.519,-11.197,-51.093,179.778,6.237,149.193
C06042=1111.524,-11.447,-51.079,179.777,6.232,149.192
C06043=1111.529,-11.696,-51.066,179.777,6.227,149.192
C06044=1111.534,-11.946,-51.053,179.777,6.223,149.191
C06045=1111.540,-12.195,-51.039,179.776,6.219,149.190
C06046=1111.544,-12.445,-51.026,179.775,6.214,149.189
C06047=1111.549,-12.695,-51.011,179.775,6.210,149.188
C06048=1111.555,-12.945,-50.998,179.774,6.205,149.187
C06049=1111.559,-13.194,-50.985,179.774,6.200,149.186
C06050=1111.565,-13.444,-50.971,179.773,6.196,149.186
C06051=1111.569,-13.693,-50.958,179.772,6.191,149.185
C06052=1111.575,-13.943,-50.945,179.772,6.186,149.184
C06053=1111.580,-14.192,-50.930,179.772,6.182,149.183
C06054=1111.585,-14.442,-50.918,179.771,6.177,149.182
C06055=1111.590,-14.691,-50.903,179.771,6.173,149.182
C06056=1111.595,-14.941,-50.891,179.770,6.169,149.181
C06057=1111.600,-15.190,-50.876,179.770,6.164,149.180
C06058=1111.605,-15.440,-50.864,179.769,6.159,149.179
C06059=1111.611,-15.690,-50.850,179.769,6.155,149.178
C06060=1111.616,-15.939,-50.836,179.768,6.150,149.177
C06061=1111.621,-16.189,-50.823,179.767,6.145,149.176
C06062=1111.626,-16.438,-50.810,179.767,6.141,149.175
C06063=1111.631,-16.688,-50.797,179.766,6.136,149.175
C06064=1111.637,-16.938,-50.783,179.766,6.131,149.174
C06065=1111.641,-17.187,-50.770,179.765,6.127,149.173
C06066=1111.646,-17.402,-50.758,179.765,6.123,149.172
C06067=1111.650,-17.616,-50.747,179.764,6.119,149.171
C06068=1111.655,-17.832,-50.735,179.764,6.115,149.171
C06069=1111.658,-18.045,-50.724,179.764,6.111,149.170
C06070=1111.663,-18.260,-50.713,179.763,6.107,149.169
C06071=1111.668,-18.474,-50.701,179.763,6.103,149.168
C06072=1111.672,-18.690,-50.690,179.762,6.099,149.168
C06073=1111.676,-18.903,-50.678,179.761,6.095,149.167
C06074=1111.682,-19.153,-50.665,179.761,6.090,149.166
C06075=1111.686,-19.403,-50.652,179.760,6.086,149.165
C06076=1111.692,-19.652,-50.639,179.760,6.081,149.164
C06077=1111.697,-19.901,-50.625,179.759,6.076,149.163
C06078=1111.702,-20.151,-50.612,179.760,6.072,149.162
C06079=1111.707,-20.401,-50.599,179.759,6.067,149.162
C06080=1111.712,-20.651,-50.586,179.759,6.063,149.161
C06081=1111.718,-20.900,-50.573,179.758,6.058,149.160
C06082=1111.722,-21.150,-50.559,179.758,6.053,149.159
C06083=1111.728,-21.399,-50.546,179.757,6.049,149.158
C06084=1111.733,-21.649,-50.534,179.757,6.044,149.157
C06085=1111.738,-21.899,-50.520,179.756,6.039,149.156
C06086=1111.743,-22.148,-50.508,179.756,6.034,149.155
C06087=1111.748,-22.397,-50.494,179.755,6.030,149.154
C06088=1111.753,-22.647,-50.481,179.755,6.025,149.153
C06089=1111.758,-22.897,-50.468,179.754,6.020,149.153
C06090=1111.763,-23.147,-50.455,179.754,6.015,149.152
C06091=1111.769,-23.396,-50.442,179.753,6.011,149.151
C06092=1111.774,-23.646,-50.429,179.753,6.006,149.150
C06093=1111.778,-23.896,-50.416,179.752,6.001,149.149
C06094=1111.784,-24.145,-50.403,179.752,5.997,149.148
C06095=1111.789,-24.395,-50.391,179.751,5.992,149.147
C06096=1111.794,-24.644,-50.377,179.751,5.987,149.146
C06097=1111.799,-24.894,-50.364,179.750,5.982,149.145
C06098=1111.805,-25.143,-50.351,179.750,5.978,149.144
C06099=1111.809,-25.393,-50.338,179.750,5.972,149.143
C06100=1111.815,-25.643,-50.325,179.750,5.968,149.142
C06101=1111.820,-25.892,-50.312,179.749,5.963,149.142
C06102=1111.825,-26.142,-50.299,179.750,5.959,149.140
C06103=1111.830,-26.391,-50.287,179.750,5.955,149.139
C06104=1111.836,-26.641,-50.274,179.750,5.950,149.138
C06105=1111.840,-26.891,-50.261,179.750,5.946,149.137
C06106=1111.845,-27.140,-50.248,179.751,5.941,149.136
C06107=1111.850,-27.390,-50.235,179.750,5.937,149.135
C06108=1111.856,-27.640,-50.222,179.750,5.933,149.135
C06109=1111.861,-27.889,-50.209,179.751,5.928,149.133
C06110=1111.866,-28.139,-50.197,179.750,5.924,149.132
C06111=1111.871,-28.388,-50.184,179.751,5.920,149.132
C06112=1111.876,-28.638,-50.170,179.751,5.915,149.130
C06113=1111.881,-28.888,-50.158,179.751,5.911,149.130
C06114=1111.887,-29.137,-50.145,179.751,5.907,149.129
C06115=1111.891,-29.387,-50.133,179.750,5.902,149.128
C06116=1111.896,-29.637,-50.120,179.751,5.898,149.127
C06117=1111.902,-29.886,-50.107,179.750,5.893,149.126
C06118=1111.907,-30.136,-50.095,179.751,5.889,149.125
C06119=1111.912,-30.386,-50.082,179.750,5.884,149.124
C06120=1111.917,-30.635,-50.069,179.750,5.880,149.123
C06121=1111.922,-30.884,-50.056,179.750,5.876,149.122
C06122=1111.927,-31.099,-50.045,179.750,5.872,149.121
C06123=1111.931,-31.314,-50.035,179.750,5.868,149.120
C06124=1111.936,-31.528,-50.024,179.749,5.865,149.120
C06125=1111.940,-31.743,-50.013,179.749,5.861,149.119
C06126=1111.944,-31.958,-50.001,179.749,5.857,149.118
C06127=1111.948,-32.172,-49.991,179.749,5.854,149.118
C06128=1111.953,-32.387,-49.980,179.749,5.850,149.117
C06129=1111.957,-32.602,-49.969,179.748,5.845,149.116
C06130=1111.963,-32.851,-49.956,179.748,5.841,149.115
C06131=1111.968,-33.100,-49.944,179.748,5.837,149.114
C06132=1111.974,-33.350,-49.931,179.747,5.832,149.113
C06133=1111.978,-33.600,-49.919,179.747,5.828,149.112
C06134=1111.984,-33.850,-49.906,179.746,5.824,149.112
C06135=1111.989,-34.099,-49.893,179.746,5.819,149.111
C06136=1111.994,-34.348,-49.881,179.746,5.814,149.110
C06137=1111.999,-34.598,-49.869,179.746,5.810,149.109
C06138=1112.004,-34.848,-49.856,179.745,5.805,149.108
C06139=1112.009,-35.098,-49.843,179.745,5.801,149.107
C06140=1112.015,-35.347,-49.830,179.744,5.796,149.106
C06141=1112.020,-35.597,-49.818,179.743,5.792,149.106
C06142=1112.025,-35.847,-49.806,179.743,5.787,149.105
C06143=1112.030,-36.097,-49.793,179.743,5.783,149.104
C06144=1112.035,-36.347,-49.781,179.743,5.778,149.103
C06145=1112.040,-36.596,-49.768,179.742,5.774,149.102
C06146=1112.045,-36.845,-49.756,179.741,5.769,149.101
C06147=1112.051,-37.094,-49.743,179.741,5.764,149.100
C06148=1112.056,-37.344,-49.731,179.740,5.760,149.099
C06149=1112.061,-37.594,-49.719,179.739,5.755,149.099
C06150=1112.066,-37.844,-49.706,179.738,5.750,149.098
C06151=1112.071,-38.094,-49.694,179.738,5.745,149.097
C06152=1112.076,-38.343,-49.681,179.738,5.740,149.096
C06153=1112.082,-38.593,-49.669,179.737,5.735,149.095
C06154=1112.087,-38.842,-49.657,179.737,5.731,149.094
C06155=1112.092,-39.092,-49.645,179.736,5.726,149.093
C06156=1112.097,-39.341,-49.632,179.735,5.721,149.093
C06157=1112.102,-39.591,-49.620,179.734,5.716,149.092
C06158=1112.108,-39.841,-49.608,179.734,5.711,149.091
C06159=1112.112,-40.091,-49.595,179.733,5.707,149.090
C06160=1112.118,-40.341,-49.583,179.732,5.701,149.089
C06161=1112.123,-40.590,-49.570,179.731,5.697,149.088
C06162=1112.128,-40.840,-49.558,179.731,5.692,149.087
C06163=1112.133,-41.089,-49.546,179.730,5.686,149.086
C06164=1112.138,-41.339,-49.534,179.729,5.682,149.086
C06165=1112.143,-41.588,-49.522,179.728,5.676,149.085
C06166=1112.149,-41.838,-49.510,179.728,5.671,149.084
C06167=1112.154,-42.087,-49.497,179.727,5.666,149.083
C06168=1112.159,-42.337,-49.485,179.726,5.661,149.082
C06169=1112.164,-42.587,-49.473,179.725,5.656,149.081
C06170=1112.170,-42.837,-49.461,179.724,5.650,149.080
C06171=1112.175,-43.087,-49.449,179.725,5.646,149.079
C06172=1112.180,-43.336,-49.437,179.725,5.641,149.078
C06173=1112.185,-43.586,-49.425,179.725,5.636,149.077
C06174=1112.190,-43.835,-49.413,179.725,5.632,149.076
C06175=1112.196,-44.085,-49.401,179.725,5.626,149.075
C06176=1112.201,-44.335,-49.389,179.726,5.622,149.074
C06177=1112.205,-44.584,-49.377,179.726,5.617,149.073
C06178=1112.211,-44.799,-49.366,179.726,5.613,149.072
C06179=1112.215,-45.014,-49.356,179.726,5.609,149.071
C06180=1112.219,-45.228,-49.346,179.726,5.605,149.070
C06181=1112.223,-45.443,-49.336,179.726,5.602,149.069
C06182=1112.228,-45.658,-49.325,179.726,5.596,149.068
C06183=1112.232,-45.872,-49.314,179.727,5.592,149.067
C06184=1112.237,-46.087,-49.304,179.727,5.589,149.066
C06185=1112.241,-46.302,-49.294,179.727,5.585,149.065
C06186=1112.246,-46.551,-49.282,179.726,5.580,149.064
C06187=1112.252,-46.801,-49.270,179.727,5.576,149.063
C06188=1112.257,-47.051,-49.258,179.727,5.570,149.062
C06189=1112.262,-47.300,-49.247,179.728,5.566,149.061
C06190=1112.267,-47.549,-49.234,179.727,5.561,149.060
C06191=1112.273,-47.799,-49.222,179.728,5.556,149.059
C06192=1112.278,-48.049,-49.211,179.728,5.552,149.057
C06193=1112.283,-48.299,-49.199,179.728,5.547,149.057
C06194=1112.288,-48.548,-49.187,179.728,5.543,149.055
C06195=1112.294,-48.798,-49.175,179.729,5.538,149.054
C06196=1112.298,-49.048,-49.163,179.729,5.533,149.053
C06197=1112.304,-49.298,-49.152,179.729,5.529,149.052
C06198=1112.309,-49.547,-49.139,179.729,5.523,149.051
C06199=1112.314,-49.797,-49.127,179.729,5.518,149.050
C06200=1112.319,-50.047,-49.116,179.729,5.514,149.049
C06201=1112.324,-50.297,-49.104,179.729,5.509,149.048
C06202=1112.330,-50.547,-49.092,179.730,5.505,149.047
C06203=1112.334,-50.796,-49.080,179.729,5.500,149.046
C06204=1112.340,-51.045,-49.068,179.730,5.495,149.045
C06205=1112.346,-51.295,-49.057,179.730,5.491,149.043
C06206=1112.350,-51.544,-49.045,179.730,5.486,149.042
C06207=1112.356,-51.794,-49.033,179.730,5.481,149.041
C06208=1112.361,-52.044,-49.022,179.731,5.476,149.040
C06209=1112.366,-52.293,-49.010,179.730,5.472,149.039
C06210=1112.371,-52.543,-48.998,179.731,5.467,149.038
C06211=1112.376,-52.793,-48.986,179.731,5.462,149.037
C06212=1112.381,-53.043,-48.974,179.730,5.458,149.036
C06213=1112.387,-53.293,-48.963,179.731,5.453,149.035
C06214=1112.393,-53.542,-48.951,179.731,5.448,149.034
C06215=1112.397,-53.791,-48.940,179.731,5.443,149.033
C06216=1112.403,-54.041,-48.928,179.732,5.439,149.032
C06217=1112.407,-54.291,-48.917,179.732,5.434,149.031
C06218=1112.413,-54.541,-48.905,179.732,5.430,149.030
C06219=1112.418,-54.791,-48.893,179.732,5.425,149.028
C06220=1112.423,-55.040,-48.881,179.732,5.420,149.027
C06221=1112.428,-55.290,-48.869,179.732,5.416,149.026
C06222=1112.433,-55.539,-48.858,179.732,5.411,149.025
C06223=1112.439,-55.789,-48.846,179.733,5.406,149.024
C06224=1112.443,-56.038,-48.835,179.733,5.401,149.023
C06225=1112.449,-56.288,-48.823,179.733,5.396,149.022
C06226=1112.454,-56.538,-48.811,179.733,5.392,149.021
C06227=1112.459,-56.788,-48.800,179.733,5.387,149.020
C06228=1112.465,-57.037,-48.788,179.733,5.382,149.019
C06229=1112.470,-57.287,-48.777,179.733,5.378,149.018
C06230=1112.475,-57.537,-48.765,179.733,5.373,149.017
C06231=1112.480,-57.786,-48.754,179.734,5.369,149.016
C06232=1112.485,-58.036,-48.742,179.734,5.364,149.015
C06233=1112.490,-58.286,-48.731,179.734,5.359,149.013
C06234=1112.495,-58.500,-48.721,179.734,5.355,149.013
C06235=1112.500,-58.715,-48.712,179.734,5.351,149.012
C06236=1112.504,-58.930,-48.702,179.734,5.347,149.011
C06237=1112.508,-59.145,-48.692,179.735,5.343,149.010
C06238=1112.513,-59.360,-48.682,179.735,5.339,149.009
C06239=1112.518,-59.574,-48.672,179.735,5.335,149.008
C06240=1112.522,-59.789,-48.662,179.735,5.330,149.007
C06241=1112.526,-60.004,-48.652,179.735,5.326,149.006
C06242=1112.531,-60.254,-48.641,179.734,5.322,149.005
C06243=1112.537,-60.503,-48.629,179.734,5.317,149.004
C06244=1112.542,-60.752,-48.618,179.733,5.311,149.003
C06245=1112.547,-61.003,-48.607,179.733,5.307,149.002
C06246=1112.552,-61.253,-48.595,179.732,5.302,149.001
C06247=1112.558,-61.502,-48.584,179.732,5.297,149.000
C06248=1112.563,-61.751,-48.573,179.731,5.291,148.999
C06249=1112.567,-62.001,-48.561,179.731,5.286,148.998
C06250=1112.573,-62.251,-48.550,179.731,5.282,148.998
C06251=1112.578,-62.501,-48.539,179.731,5.277,148.996
C06252=1112.584,-62.751,-48.527,179.730,5.271,148.995
C06253=1112.589,-63.000,-48.516,179.729,5.266,148.995
C06254=1112.593,-63.250,-48.505,179.729,5.261,148.993
C06255=1112.599,-63.499,-48.493,179.728,5.256,148.992
C06256=1112.604,-63.749,-48.483,179.728,5.251,148.992
C06257=1112.610,-63.999,-48.471,179.728,5.246,148.990
C06258=1112.614,-64.249,-48.460,179.728,5.241,148.989
C06259=1112.620,-64.498,-48.449,179.727,5.235,148.988
C06260=1112.625,-64.748,-48.437,179.727,5.230,148.987
C06261=1112.630,-64.998,-48.426,179.726,5.225,148.986
C06262=1112.635,-65.247,-48.415,179.727,5.220,148.985
C06263=1112.641,-65.497,-48.404,179.726,5.215,148.984
C06264=1112.646,-65.747,-48.393,179.726,5.210,148.983
C06265=1112.651,-65.996,-48.382,179.725,5.205,148.982
C06266=1112.657,-66.247,-48.371,179.726,5.200,148.981
C06267=1112.662,-66.496,-48.359,179.725,5.195,148.980
C06268=1112.667,-66.745,-48.348,179.725,5.189,148.979
C06269=1112.673,-66.996,-48.337,179.724,5.184,148.978
C06270=1112.677,-67.245,-48.326,179.724,5.179,148.977
C06271=1112.683,-67.495,-48.316,179.725,5.174,148.976
C06272=1112.688,-67.744,-48.305,179.724,5.168,148.975
C06273=1112.694,-67.994,-48.293,179.724,5.163,148.974
C06274=1112.699,-68.244,-48.282,179.723,5.158,148.973
C06275=1112.703,-68.494,-48.271,179.723,5.153,148.972
C06276=1112.709,-68.743,-48.261,179.724,5.148,148.970
C06277=1112.714,-68.993,-48.249,179.723,5.143,148.969
C06278=1112.719,-69.243,-48.238,179.723,5.137,148.968
C06279=1112.725,-69.492,-48.228,179.723,5.132,148.967
C06280=1112.729,-69.742,-48.216,179.723,5.128,148.966
C06281=1112.735,-69.991,-48.206,179.723,5.122,148.965
C06282=1112.740,-70.241,-48.194,179.723,5.117,148.964
C06283=1112.745,-70.492,-48.184,179.722,5.111,148.963
C06284=1112.751,-70.740,-48.173,179.722,5.107,148.962
C06285=1112.756,-70.991,-48.162,179.722,5.101,148.961
C06286=1112.761,-71.240,-48.152,179.722,5.096,148.959
C06287=1112.767,-71.490,-48.140,179.722,5.091,148.958
C06288=1112.772,-71.740,-48.130,179.722,5.086,148.957
C06289=1112.777,-71.989,-48.119,179.722,5.081,148.956
C06290=1112.782,-72.205,-48.109,179.722,5.076,148.955
C06291=1112.786,-72.419,-48.100,179.721,5.072,148.954
C06292=1112.790,-72.634,-48.091,179.722,5.067,148.953
C06293=1112.795,-72.848,-48.081,179.722,5.063,148.952
C06294=1112.799,-73.063,-48.073,179.722,5.059,148.951
C06295=1112.804,-73.279,-48.063,179.722,5.054,148.950
C06296=1112.809,-73.493,-48.054,179.722,5.050,148.949
C06297=1112.814,-73.709,-48.044,179.722,5.045,148.949
C06298=1112.819,-73.958,-48.033,179.722,5.040,148.947
C06299=1112.824,-74.208,-48.023,179.722,5.035,148.946
C06300=1112.829,-74.457,-48.013,179.722,5.030,148.945
C06301=1112.834,-74.707,-48.001,179.722,5.025,148.944
C06302=1112.840,-74.957,-47.991,179.722,5.019,148.943
C06303=1112.845,-75.207,-47.981,179.722,5.014,148.942
C06304=1112.850,-75.456,-47.970,179.723,5.009,148.940
C06305=1112.855,-75.706,-47.959,179.722,5.003,148.939
C06306=1112.861,-75.955,-47.949,179.722,4.998,148.938
C06307=1112.865,-76.205,-47.938,179.722,4.993,148.937
C06308=1112.871,-76.455,-47.927,179.722,4.988,148.936
C06309=1112.877,-76.705,-47.916,179.722,4.983,148.935
C06310=1112.882,-76.955,-47.906,179.722,4.978,148.934
C06311=1112.887,-77.204,-47.895,179.722,4.973,148.932
C06312=1112.893,-77.454,-47.884,179.723,4.968,148.931
C06313=1112.898,-77.704,-47.874,179.723,4.962,148.930
C06314=1112.903,-77.954,-47.864,179.723,4.957,148.929
C06315=1112.908,-78.203,-47.853,179.723,4.952,148.928
C06316=1112.913,-78.453,-47.842,179.723,4.947,148.927
C06317=1112.919,-78.702,-47.832,179.723,4.942,148.925
C06318=1112.924,-78.953,-47.821,179.724,4.937,148.924
C06319=1112.930,-79.202,-47.811,179.724,4.932,148.923
C06320=1112.934,-79.452,-47.800,179.724,4.926,148.922
C06321=1112.940,-79.701,-47.790,179.724,4.921,148.921
C06322=1112.945,-79.951,-47.779,179.724,4.916,148.919
C06323=1112.950,-80.201,-47.769,179.725,4.911,148.918
C06324=1112.956,-80.451,-47.759,179.725,4.905,148.917
C06325=1112.961,-80.701,-47.748,179.725,4.900,148.916
C06326=1112.966,-80.950,-47.738,179.725,4.895,148.915
C06327=1112.971,-81.199,-47.728,179.726,4.890,148.913
C06328=1112.976,-81.449,-47.717,179.726,4.886,148.912
C06329=1112.982,-81.699,-47.707,179.726,4.880,148.911
C06330=1112.987,-81.949,-47.696,179.727,4.875,148.910
C06331=1112.992,-82.199,-47.686,179.727,4.870,148.909
C06332=1112.998,-82.448,-47.676,179.727,4.865,148.907
C06333=1113.003,-82.698,-47.665,179.727,4.860,148.906
C06334=1113.009,-82.948,-47.655,179.727,4.855,148.905
C06335=1113.014,-83.198,-47.644,179.727,4.850,148.904
C06336=1113.019,-83.447,-47.634,179.728,4.844,148.903
C06337=1113.024,-83.696,-47.624,179.728,4.839,148.901
C06338=1113.029,-83.947,-47.613,179.729,4.835,148.900
C06339=1113.034,-84.196,-47.603,179.729,4.829,148.899
C06340=1113.040,-84.446,-47.593,179.729,4.824,148.898
C06341=1113.045,-84.696,-47.582,179.730,4.819,148.897
C06342=1113.051,-84.946,-47.572,179.730,4.814,148.895
C06343=1113.056,-85.195,-47.562,179.730,4.809,148.894
C06344=1113.060,-85.445,-47.552,179.731,4.804,148.893
C06345=1113.066,-85.695,-47.542,179.731,4.799,148.892
C06346=1113.075,-86.111,-47.525,179.732,4.791,148.890
C06347=1113.083,-86.528,-47.508,179.732,4.782,148.888
C06348=1113.093,-86.944,-47.491,179.733,4.774,148.886
C06349=1113.102,-87.361,-47.474,179.734,4.766,148.884
C06350=1113.107,-87.664,-47.462,179.734,4.759,148.882
C06351=1113.113,-87.913,-47.451,179.734,4.754,148.881
C06352=1113.118,-88.163,-47.441,179.735,4.750,148.880
C06353=1113.124,-88.414,-47.431,179.736,4.744,148.878
C06354=1113.129,-88.663,-47.422,179.736,4.739,148.877
C06355=1113.134,-88.913,-47.411,179.737,4.735,148.876
C06356=1113.139,-89.163,-47.401,179.737,4.730,148.875
C06357=1113.145,-89.412,-47.391,179.737,4.725,148.874
C06358=1113.150,-89.662,-47.380,179.737,4.719,148.873
C06359=1113.155,-89.912,-47.371,179.738,4.715,148.871
C06360=1113.161,-90.161,-47.360,179.739,4.709,148.870
C06361=1113.166,-90.411,-47.351,179.739,4.705,148.869
C06362=1113.171,-90.661,-47.341,179.740,4.700,148.868
C06363=1113.176,-90.911,-47.331,179.740,4.695,148.866
C06364=1113.182,-91.160,-47.320,179.741,4.690,148.865
C06365=1113.187,-91.410,-47.310,179.741,4.685,148.864
C06366=1113.192,-91.660,-47.300,179.741,4.680,148.863
C06367=1113.198,-91.910,-47.291,179.742,4.675,148.861
C06368=1113.203,-92.160,-47.281,179.743,4.670,148.860
C06369=1113.208,-92.409,-47.271,179.743,4.666,148.859
C06370=1113.213,-92.659,-47.260,179.744,4.661,148.858
C06371=1113.219,-92.909,-47.250,179.744,4.656,148.857
C06372=1113.224,-93.158,-47.241,179.745,4.651,148.855
C06373=1113.229,-93.408,-47.231,179.745,4.646,148.854
C06374=1113.234,-93.658,-47.221,179.746,4.641,148.853
C06375=1113.239,-93.907,-47.211,179.746,4.636,148.852
C06376=1113.245,-94.158,-47.201,179.747,4.632,148.850
C06377=1113.251,-94.407,-47.191,179.747,4.627,148.849
C06378=1113.256,-94.656,-47.182,179.748,4.622,148.848
C06379=1113.261,-94.907,-47.171,179.748,4.617,148.847
C06380=1113.267,-95.157,-47.162,179.748,4.612,148.846
C06381=1113.271,-95.406,-47.152,179.749,4.607,148.845
C06382=1113.277,-95.656,-47.142,179.749,4.603,148.843
C06383=1113.283,-95.906,-47.132,179.750,4.597,148.842
C06384=1113.287,-96.156,-47.122,179.750,4.592,148.841
C06385=1113.293,-96.405,-47.112,179.751,4.588,148.840
C06386=1113.298,-96.655,-47.103,179.750,4.583,148.839
C06387=1113.304,-96.905,-47.093,179.751,4.578,148.838
C06388=1113.309,-97.154,-47.083,179.751,4.573,148.836
C06389=1113.314,-97.404,-47.074,179.752,4.569,148.835
C06390=1113.319,-97.654,-47.063,179.752,4.563,148.834
C06391=1113.324,-97.903,-47.054,179.752,4.558,148.833
C06392=1113.330,-98.154,-47.044,179.752,4.553,148.832
C06393=1113.336,-98.403,-47.034,179.753,4.549,148.830
C06394=1113.341,-98.653,-47.025,179.753,4.544,148.829
C06395=1113.346,-98.903,-47.015,179.753,4.538,148.828
C06396=1113.351,-99.152,-47.005,179.754,4.533,148.827
C06397=1113.357,-99.403,-46.995,179.754,4.529,148.826
C06398=1113.361,-99.617,-46.987,179.754,4.524,148.825
C06399=1113.366,-99.832,-46.979,179.755,4.520,148.824
C06400=1113.370,-100.047,-46.971,179.755,4.516,148.823
C06401=1113.375,-100.262,-46.962,179.756,4.512,148.822
C06402=1113.380,-100.477,-46.954,179.756,4.507,148.820
C06403=1113.384,-100.692,-46.945,179.756,4.503,148.819
C06404=1113.388,-100.907,-46.937,179.756,4.499,148.819
C06405=1113.393,-101.122,-46.930,179.757,4.495,148.818
C06406=1113.399,-101.372,-46.919,179.757,4.490,148.816
C06407=1113.403,-101.622,-46.910,179.757,4.484,148.815
C06408=1113.409,-101.872,-46.900,179.757,4.479,148.814
C06409=1113.414,-102.121,-46.891,179.758,4.475,148.813
C06410=1113.420,-102.371,-46.881,179.758,4.470,148.812
C06411=1113.425,-102.621,-46.872,179.759,4.465,148.810
C06412=1113.430,-102.870,-46.862,179.759,4.460,148.809
C06413=1113.436,-103.120,-46.853,179.759,4.454,148.808
C06414=1113.441,-103.370,-46.843,179.760,4.450,148.807
C06415=1113.446,-103.620,-46.834,179.760,4.445,148.806
C06416=1113.452,-103.869,-46.823,179.760,4.440,148.804
C06417=1113.457,-104.120,-46.814,179.761,4.435,148.803
C06418=1113.462,-104.369,-46.804,179.761,4.429,148.802
C06419=1113.467,-104.619,-46.795,179.761,4.424,148.801
C06420=1113.472,-104.868,-46.785,179.762,4.420,148.800
C06421=1113.478,-105.119,-46.776,179.762,4.415,148.798
C06422=1113.483,-105.368,-46.767,179.762,4.410,148.797
C06423=1113.489,-105.618,-46.757,179.763,4.404,148.796
C06424=1113.494,-105.868,-46.748,179.763,4.399,148.795
C06425=1113.499,-106.117,-46.738,179.764,4.395,148.794
C06426=1113.505,-106.367,-46.729,179.764,4.390,148.792
C06427=1113.510,-106.617,-46.720,179.764,4.385,148.791
C06428=1113.515,-106.867,-46.710,179.764,4.379,148.790
C06429=1113.521,-107.116,-46.701,179.765,4.374,148.789
C06430=1113.526,-107.366,-46.692,179.765,4.369,148.788
C06431=1113.531,-107.616,-46.682,179.765,4.364,148.786
C06432=1113.537,-107.866,-46.673,179.766,4.360,148.785
C06433=1113.542,-108.116,-46.664,179.766,4.354,148.784
C06434=1113.547,-108.365,-46.654,179.767,4.349,148.783
C06435=1113.553,-108.615,-46.645,179.767,4.344,148.781
C06436=1113.558,-108.865,-46.636,179.767,4.339,148.780
C06437=1113.563,-109.114,-46.626,179.768,4.333,148.779
C06438=1113.568,-109.364,-46.617,179.768,4.328,148.778
C06439=1113.574,-109.614,-46.608,179.768,4.323,148.777
C06440=1113.580,-109.864,-46.598,179.769,4.319,148.775
C06441=1113.584,-110.113,-46.589,179.769,4.314,148.774
C06442=1113.590,-110.363,-46.580,179.769,4.308,148.773
C06443=1113.595,-110.613,-46.570,179.770,4.303,148.772
C06444=1113.601,-110.863,-46.562,179.770,4.298,148.771
C06445=1113.605,-111.112,-46.552,179.770,4.293,148.769
C06446=1113.611,-111.362,-46.543,179.770,4.288,148.768
C06447=1113.617,-111.613,-46.534,179.771,4.283,148.767
C06448=1113.622,-111.862,-46.525,179.771,4.277,148.766
C06449=1113.627,-112.112,-46.516,179.771,4.272,148.765
C06450=1113.632,-112.362,-46.506,179.771,4.267,148.763
C06451=1113.638,-112.612,-46.497,179.773,4.262,148.762
C06452=1113.643,-112.861,-46.488,179.773,4.257,148.761
C06453=1113.648,-113.111,-46.479,179.773,4.252,148.759
C06454=1113.653,-113.326,-46.471,179.773,4.247,148.759
C06455=1113.657,-113.541,-46.463,179.774,4.243,148.757
C06456=1113.662,-113.756,-46.455,179.774,4.238,148.756
C06457=1113.667,-113.971,-46.448,179.774,4.234,148.755
C06458=1113.671,-114.187,-46.440,179.775,4.230,148.754
C06459=1113.676,-114.401,-46.431,179.775,4.225,148.753
C06460=1113.680,-114.616,-46.424,179.775,4.221,148.752
C06461=1113.685,-114.832,-46.416,179.775,4.216,148.751
C06462=1113.690,-115.081,-46.407,179.775,4.211,148.750
C06463=1113.696,-115.331,-46.398,179.776,4.206,148.749
C06464=1113.702,-115.581,-46.389,179.777,4.201,148.747
C06465=1113.707,-115.831,-46.380,179.777,4.196,148.746
C06466=1113.712,-116.081,-46.371,179.778,4.190,148.745
C06467=1113.717,-116.331,-46.362,179.778,4.185,148.744
C06468=1113.722,-116.579,-46.353,179.778,4.180,148.742
C06469=1113.728,-116.829,-46.344,179.778,4.175,148.741
C06470=1113.734,-117.079,-46.334,179.779,4.170,148.740
C06471=1113.739,-117.329,-46.326,179.779,4.165,148.739
C06472=1113.744,-117.579,-46.317,179.780,4.159,148.737
C06473=1113.749,-117.829,-46.308,179.780,4.154,148.736
C06474=1113.754,-118.079,-46.299,179.780,4.149,148.735
C06475=1113.760,-118.328,-46.290,179.780,4.143,148.734
C06476=1113.765,-118.578,-46.281,179.780,4.138,148.732
C06477=1113.771,-118.828,-46.272,179.781,4.132,148.731
C06478=1113.776,-119.078,-46.263,179.781,4.127,148.730
C06479=1113.781,-119.328,-46.254,179.782,4.122,148.729
C06480=1113.787,-119.578,-46.245,179.782,4.117,148.727
C06481=1113.792,-119.827,-46.237,179.782,4.111,148.726
C06482=1113.798,-120.077,-46.229,179.782,4.106,148.725
C06483=1113.803,-120.327,-46.220,179.783,4.101,148.723
C06484=1113.808,-120.577,-46.211,179.784,4.096,148.722
C06485=1113.813,-120.827,-46.202,179.784,4.090,148.721
C06486=1113.818,-121.077,-46.193,179.784,4.085,148.720
C06487=1113.824,-121.326,-46.184,179.785,4.080,148.718
C06488=1113.829,-121.576,-46.176,179.785,4.074,148.717
C06489=1113.835,-121.825,-46.167,179.786,4.069,148.716
C06490=1113.840,-122.075,-46.158,179.786,4.064,148.715
C06491=1113.846,-122.325,-46.148,179.787,4.059,148.713
C06492=1113.851,-122.575,-46.140,179.786,4.053,148.712
C06493=1113.857,-122.825,-46.132,179.787,4.047,148.711
C06494=1113.862,-123.075,-46.123,179.787,4.042,148.710
C06495=1113.867,-123.325,-46.114,179.788,4.037,148.708
C06496=1113.873,-123.574,-46.105,179.788,4.032,148.707
C06497=1113.878,-123.824,-46.096,179.788,4.026,148.706
C06498=1113.883,-124.074,-46.087,179.789,4.021,148.704
C06499=1113.889,-124.324,-46.079,179.789,4.016,148.703
C06500=1113.895,-124.573,-46.071,179.789,4.010,148.702
C06501=1113.899,-124.823,-46.062,179.789,4.005,148.701
C06502=1113.904,-125.073,-46.054,179.790,3.999,148.699
C06503=1113.910,-125.323,-46.045,179.791,3.994,148.698
C06504=1113.915,-125.572,-46.037,179.791,3.989,148.697
C06505=1113.921,-125.822,-46.028,179.792,3.983,148.695
C06506=1113.926,-126.072,-46.019,179.792,3.978,148.694
C06507=1113.931,-126.322,-46.011,179.792,3.972,148.693
C06508=1113.937,-126.572,-46.002,179.793,3.966,148.691
C06509=1113.942,-126.821,-45.993,179.793,3.961,148.690
C06510=1113.947,-127.037,-45.986,179.793,3.956,148.689
C06511=1113.951,-127.251,-45.979,179.794,3.952,148.688
C06512=1113.956,-127.467,-45.972,179.794,3.947,148.687
C06513=1113.961,-127.682,-45.964,179.795,3.943,148.685
C06514=1113.966,-127.897,-45.957,179.794,3.938,148.684
C06515=1113.970,-128.112,-45.950,179.795,3.933,148.683
C06516=1113.975,-128.327,-45.942,179.796,3.928,148.682
C06517=1113.980,-128.543,-45.935,179.795,3.923,148.681
C06518=1113.556,-128.534,-45.960,179.803,3.928,148.680
C06519=1113.551,-128.319,-45.968,179.802,3.932,148.681
C06520=1113.547,-128.103,-45.976,179.802,3.937,148.682
C06521=1113.542,-127.887,-45.983,179.802,3.942,148.683
C06522=1113.538,-127.672,-45.990,179.801,3.946,148.684
C06523=1113.533,-127.457,-45.997,179.802,3.951,148.685
C06524=1113.528,-127.242,-46.005,179.801,3.956,148.686
C06525=1113.524,-127.027,-46.012,179.800,3.961,148.688
C06526=1113.519,-126.812,-46.020,179.801,3.965,148.689
C06527=1113.514,-126.562,-46.029,179.800,3.971,148.690
C06528=1113.508,-126.313,-46.036,179.799,3.976,148.691
C06529=1113.503,-126.063,-46.045,179.799,3.981,148.693
C06530=1113.498,-125.813,-46.054,179.798,3.987,148.694
C06531=1113.492,-125.564,-46.063,179.798,3.992,148.695
C06532=1113.487,-125.313,-46.071,179.798,3.998,148.697
C06533=1113.481,-125.063,-46.080,179.797,4.004,148.698
C06534=1113.476,-124.814,-46.089,179.797,4.009,148.699
C06535=1113.471,-124.564,-46.098,179.797,4.014,148.700
C06536=1113.465,-124.315,-46.106,179.796,4.020,148.702
C06537=1113.460,-124.064,-46.114,179.796,4.025,148.703
C06538=1113.455,-123.814,-46.123,179.795,4.030,148.704
C06539=1113.450,-123.564,-46.132,179.795,4.035,148.706
C06540=1113.444,-123.315,-46.141,179.795,4.041,148.707
C06541=1113.439,-123.065,-46.150,179.795,4.047,148.708
C06542=1113.433,-122.816,-46.158,179.794,4.052,148.710
C06543=1113.428,-122.566,-46.167,179.794,4.057,148.711
C06544=1113.423,-122.316,-46.176,179.793,4.062,148.712
C06545=1113.417,-122.066,-46.184,179.793,4.068,148.713
C06546=1113.412,-121.816,-46.193,179.792,4.073,148.715
C06547=1113.407,-121.566,-46.202,179.792,4.078,148.716
C06548=1113.402,-121.317,-46.211,179.792,4.083,148.717
C06549=1113.396,-121.067,-46.220,179.791,4.089,148.718
C06550=1113.391,-120.818,-46.228,179.790,4.094,148.720
C06551=1113.385,-120.568,-46.237,179.791,4.100,148.721
C06552=1113.380,-120.318,-46.247,179.791,4.105,148.722
C06553=1113.374,-120.068,-46.255,179.790,4.111,148.723
C06554=1113.369,-119.818,-46.264,179.789,4.116,148.725
C06555=1113.364,-119.568,-46.273,179.789,4.121,148.726
C06556=1113.358,-119.319,-46.282,179.789,4.126,148.727
C06557=1113.353,-119.069,-46.291,179.789,4.132,148.728
C06558=1113.348,-118.819,-46.300,179.788,4.137,148.730
C06559=1113.343,-118.569,-46.309,179.788,4.142,148.731
C06560=1113.338,-118.319,-46.317,179.787,4.147,148.732
C06561=1113.332,-118.069,-46.327,179.787,4.153,148.734
C06562=1113.327,-117.819,-46.336,179.787,4.158,148.735
C06563=1113.321,-117.570,-46.344,179.786,4.163,148.736
C06564=1113.316,-117.320,-46.353,179.786,4.168,148.737
C06565=1113.310,-117.071,-46.362,179.785,4.174,148.739
C06566=1113.305,-116.821,-46.371,179.785,4.179,148.740
C06567=1113.299,-116.571,-46.381,179.785,4.184,148.741
C06568=1113.294,-116.321,-46.389,179.785,4.189,148.742
C06569=1113.289,-116.071,-46.398,179.784,4.194,148.744
C06570=1113.284,-115.822,-46.408,179.784,4.199,148.745
C06571=1113.279,-115.572,-46.417,179.783,4.205,148.746
C06572=1113.273,-115.322,-46.426,179.783,4.210,148.747
C06573=1113.267,-115.072,-46.435,179.783,4.215,148.749
C06574=1113.262,-114.823,-46.444,179.782,4.220,148.750
C06575=1113.257,-114.607,-46.451,179.782,4.224,148.751
C06576=1113.253,-114.392,-46.459,179.781,4.229,148.752
C06577=1113.249,-114.177,-46.468,179.781,4.234,148.753
C06578=1113.244,-113.962,-46.475,179.781,4.238,148.754
C06579=1113.239,-113.747,-46.483,179.781,4.243,148.755
C06580=1113.235,-113.533,-46.491,179.781,4.247,148.756
C06581=1113.230,-113.317,-46.499,179.780,4.251,148.757
C06582=1113.225,-113.102,-46.507,179.780,4.256,148.758
C06583=1113.220,-112.852,-46.516,179.780,4.261,148.759
C06584=1113.215,-112.603,-46.525,179.779,4.266,148.761
C06585=1113.210,-112.352,-46.535,179.779,4.272,148.762
C06586=1113.204,-112.103,-46.544,179.778,4.277,148.763
C06587=1113.199,-111.853,-46.553,179.778,4.281,148.765
C06588=1113.193,-111.603,-46.562,179.777,4.286,148.766
C06589=1113.188,-111.353,-46.572,179.777,4.292,148.767
C06590=1113.183,-111.104,-46.580,179.777,4.297,148.768
C06591=1113.178,-110.854,-46.589,179.777,4.302,148.769
C06592=1113.172,-110.604,-46.599,179.776,4.307,148.771
C06593=1113.167,-110.355,-46.608,179.776,4.312,148.772
C06594=1113.162,-110.105,-46.617,179.776,4.317,148.773
C06595=1113.156,-109.855,-46.627,179.776,4.322,148.774
C06596=1113.151,-109.606,-46.636,179.775,4.328,148.775
C06597=1113.146,-109.356,-46.645,179.775,4.332,148.777
C06598=1113.140,-109.106,-46.655,179.774,4.337,148.778
C06599=1113.135,-108.856,-46.664,179.774,4.342,148.779
C06600=1113.130,-108.607,-46.673,179.774,4.347,148.780
C06601=1113.124,-108.356,-46.683,179.773,4.353,148.782
C06602=1113.119,-108.107,-46.692,179.773,4.358,148.783
C06603=1113.114,-107.856,-46.702,179.773,4.363,148.784
C06604=1113.109,-107.606,-46.711,179.772,4.369,148.785
C06605=1113.104,-107.357,-46.721,179.771,4.373,148.786
C06606=1113.098,-107.107,-46.730,179.771,4.378,148.788
C06607=1113.093,-106.857,-46.739,179.771,4.383,148.789
C06608=1113.088,-106.608,-46.749,179.771,4.388,148.790
C06609=1113.082,-106.358,-46.758,179.770,4.393,148.791
C06610=1113.077,-106.109,-46.768,179.770,4.399,148.792
C06611=1113.071,-105.858,-46.777,179.769,4.403,148.794
C06612=1113.066,-105.609,-46.786,179.769,4.408,148.795
C06613=1113.061,-105.359,-46.796,179.769,4.413,148.796
C06614=1113.055,-105.109,-46.805,179.769,4.418,148.797
C06615=1113.050,-104.860,-46.815,179.768,4.424,148.798
C06616=1113.044,-104.610,-46.824,179.768,4.429,148.800
C06617=1113.039,-104.361,-46.834,179.767,4.433,148.801
C06618=1113.034,-104.110,-46.843,179.767,4.438,148.802
C06619=1113.029,-103.861,-46.853,179.767,4.443,148.803
C06620=1113.023,-103.610,-46.863,179.767,4.449,148.804
C06621=1113.018,-103.360,-46.872,179.766,4.454,148.806
C06622=1113.013,-103.111,-46.882,179.766,4.458,148.807
C06623=1113.007,-102.861,-46.891,179.765,4.463,148.808
C06624=1113.003,-102.612,-46.901,179.765,4.468,148.809
C06625=1112.997,-102.362,-46.911,179.765,4.474,148.810
C06626=1112.992,-102.112,-46.920,179.765,4.479,148.812
C06627=1112.986,-101.863,-46.930,179.764,4.483,148.813
C06628=1112.981,-101.613,-46.939,179.764,4.488,148.814
C06629=1112.976,-101.363,-46.949,179.763,4.493,148.815
C06630=1112.971,-101.113,-46.958,179.763,4.499,148.816
C06631=1112.963,-100.757,-46.972,179.763,4.505,148.818
C06632=1112.955,-100.399,-46.986,179.762,4.512,148.820
C06633=1112.948,-100.041,-47.000,179.762,4.520,148.821
C06634=1112.940,-99.684,-47.014,179.761,4.526,148.823
C06635=1112.935,-99.435,-47.024,179.761,4.531,148.824
C06636=1112.929,-99.185,-47.033,179.761,4.537,148.825
C06637=1112.924,-98.935,-47.043,179.760,4.541,148.827
C06638=1112.919,-98.685,-47.052,179.760,4.546,148.828
C06639=1112.914,-98.435,-47.063,179.760,4.551,148.829
C06640=1112.908,-98.186,-47.073,179.759,4.556,148.830
C06641=1112.903,-97.936,-47.082,179.759,4.561,148.831
C06642=1112.897,-97.686,-47.092,179.758,4.566,148.833
C06643=1112.893,-97.437,-47.102,179.758,4.571,148.834
C06644=1112.887,-97.187,-47.111,179.758,4.576,148.835
C06645=1112.882,-96.937,-47.122,179.757,4.581,148.836
C06646=1112.877,-96.687,-47.131,179.757,4.586,148.837
C06647=1112.869,-96.364,-47.144,179.757,4.592,148.839
C06648=1112.863,-96.042,-47.157,179.756,4.599,148.840
C06649=1112.856,-95.720,-47.170,179.756,4.605,148.842
C06650=1112.849,-95.397,-47.182,179.755,4.611,148.844
C06651=1112.843,-95.148,-47.192,179.755,4.616,148.845
C06652=1112.839,-94.898,-47.202,179.755,4.621,148.846
C06653=1112.833,-94.648,-47.212,179.755,4.626,148.847
C06654=1112.827,-94.398,-47.222,179.754,4.631,148.848
C06655=1112.823,-94.149,-47.231,179.754,4.636,148.849
C06656=1112.818,-93.899,-47.242,179.752,4.640,148.851
C06657=1112.812,-93.649,-47.252,179.752,4.646,148.852
C06658=1112.807,-93.399,-47.261,179.751,4.650,148.853
C06659=1112.801,-93.150,-47.271,179.751,4.655,148.854
C06660=1112.796,-92.900,-47.282,179.751,4.660,148.855
C06661=1112.791,-92.650,-47.292,179.750,4.665,148.857
C06662=1112.786,-92.401,-47.302,179.750,4.670,148.858
C06663=1112.780,-92.150,-47.311,179.749,4.674,148.859
C06664=1112.775,-91.900,-47.322,179.748,4.680,148.860
C06665=1112.770,-91.651,-47.331,179.748,4.684,148.862
C06666=1112.764,-91.401,-47.342,179.747,4.689,148.863
C06667=1112.759,-91.152,-47.352,179.747,4.694,148.864
C06668=1112.755,-90.902,-47.362,179.747,4.699,148.865
C06669=1112.749,-90.652,-47.371,179.746,4.704,148.866
C06670=1112.743,-90.402,-47.382,179.746,4.709,148.868
C06671=1112.737,-90.153,-47.392,179.745,4.713,148.869
C06672=1112.733,-89.903,-47.402,179.745,4.719,148.870
C06673=1112.728,-89.653,-47.412,179.744,4.724,148.871
C06674=1112.722,-89.404,-47.422,179.744,4.728,148.873
C06675=1112.717,-89.153,-47.433,179.743,4.733,148.874
C06676=1112.712,-88.904,-47.442,179.743,4.739,148.875
C06677=1112.707,-88.655,-47.453,179.743,4.743,148.876
C06678=1112.701,-88.404,-47.462,179.742,4.748,148.877
C06679=1112.696,-88.154,-47.473,179.742,4.754,148.879
C06680=1112.690,-87.905,-47.483,179.741,4.758,148.880
C06681=1112.685,-87.656,-47.492,179.741,4.763,148.881
C06682=1112.680,-87.405,-47.503,179.741,4.768,148.882
C06683=1112.675,-87.190,-47.512,179.740,4.772,148.883
C06684=1112.671,-86.975,-47.521,179.739,4.777,148.884
C06685=1112.667,-86.761,-47.529,179.740,4.781,148.885
C06686=1112.662,-86.545,-47.538,179.739,4.786,148.886
C06687=1112.657,-86.331,-47.547,179.739,4.790,148.887
C06688=1112.653,-86.116,-47.557,179.738,4.794,148.889
C06689=1112.649,-85.902,-47.565,179.738,4.799,148.890
C06690=1112.644,-85.686,-47.574,179.738,4.803,148.890
C06691=1112.639,-85.437,-47.584,179.737,4.808,148.892
C06692=1112.633,-85.187,-47.594,179.737,4.813,148.893
C06693=1112.628,-84.937,-47.605,179.736,4.818,148.894
C06694=1112.623,-84.688,-47.615,179.736,4.823,148.895
C06695=1112.617,-84.438,-47.625,179.736,4.828,148.897
C06696=1112.612,-84.188,-47.636,179.736,4.833,148.898
C06697=1112.607,-83.938,-47.646,179.736,4.838,148.899
C06698=1112.601,-83.689,-47.656,179.736,4.843,148.900
C06699=1112.597,-83.439,-47.666,179.735,4.848,148.901
C06700=1112.591,-83.189,-47.676,179.734,4.853,148.903
C06701=1112.586,-82.939,-47.687,179.734,4.858,148.904
C06702=1112.581,-82.689,-47.697,179.734,4.864,148.905
C06703=1112.575,-82.440,-47.707,179.734,4.869,148.906
C06704=1112.570,-82.190,-47.718,179.733,4.874,148.907
C06705=1112.565,-81.941,-47.729,179.733,4.879,148.909
C06706=1112.560,-81.690,-47.739,179.733,4.884,148.910
C06707=1112.554,-81.441,-47.749,179.733,4.889,148.911
C06708=1112.548,-81.191,-47.760,179.733,4.895,148.912
C06709=1112.543,-80.941,-47.770,179.733,4.900,148.913
C06710=1112.538,-80.692,-47.780,179.732,4.904,148.915
C06711=1112.533,-80.442,-47.792,179.731,4.910,148.916
C06712=1112.528,-80.192,-47.802,179.731,4.915,148.917
C06713=1112.523,-79.942,-47.812,179.731,4.920,148.918
C06714=1112.517,-79.693,-47.823,179.731,4.925,148.919
C06715=1112.511,-79.443,-47.833,179.731,4.930,148.921
C06716=1112.507,-79.193,-47.844,179.730,4.935,148.922
C06717=1112.501,-78.944,-47.854,179.730,4.940,148.923
C06718=1112.496,-78.694,-47.865,179.730,4.946,148.924
C06719=1112.491,-78.444,-47.875,179.730,4.951,148.925
C06720=1112.486,-78.194,-47.886,179.730,4.956,148.926
C06721=1112.480,-77.945,-47.897,179.730,4.961,148.928
C06722=1112.475,-77.695,-47.907,179.729,4.966,148.929
C06723=1112.470,-77.445,-47.917,179.729,4.971,148.930
C06724=1112.464,-77.196,-47.928,179.729,4.976,148.931
C06725=1112.459,-76.946,-47.939,179.729,4.982,148.932
C06726=1112.454,-76.696,-47.949,179.729,4.987,148.934
C06727=1112.449,-76.446,-47.960,179.729,4.992,148.935
C06728=1112.443,-76.197,-47.971,179.729,4.997,148.936
C06729=1112.438,-75.947,-47.981,179.728,5.002,148.937
C06730=1112.433,-75.697,-47.991,179.729,5.008,148.938
C06731=1112.428,-75.448,-48.003,179.729,5.013,148.939
C06732=1112.423,-75.198,-48.013,179.729,5.018,148.940
C06733=1112.417,-74.948,-48.024,179.729,5.023,148.941
C06734=1112.412,-74.699,-48.035,179.729,5.028,148.943
C06735=1112.407,-74.449,-48.046,179.729,5.033,148.944
C06736=1112.401,-74.199,-48.056,179.728,5.039,148.945
C06737=1112.396,-73.949,-48.067,179.728,5.044,148.946
C06738=1112.391,-73.699,-48.078,179.728,5.049,148.947
C06739=1112.386,-73.485,-48.087,179.729,5.054,148.948
C06740=1112.382,-73.269,-48.097,179.728,5.058,148.949
C06741=1112.377,-73.056,-48.106,179.729,5.062,148.950
C06742=1112.373,-72.840,-48.115,179.728,5.066,148.951
C06743=1112.368,-72.626,-48.125,179.728,5.071,148.952
C06744=1112.364,-72.411,-48.133,179.728,5.075,148.953
C06745=1112.360,-72.196,-48.143,179.728,5.080,148.954
C06746=1112.354,-71.981,-48.152,179.729,5.085,148.955
C06747=1112.350,-71.732,-48.164,179.729,5.090,148.956
C06748=1112.344,-71.482,-48.174,179.728,5.095,148.957
C06749=1112.339,-71.232,-48.184,179.729,5.100,148.958
C06750=1112.334,-70.982,-48.196,179.729,5.105,148.959
C06751=1112.328,-70.732,-48.206,179.729,5.110,148.961
C06752=1112.323,-70.483,-48.218,179.728,5.115,148.962
C06753=1112.318,-70.234,-48.229,179.729,5.121,148.963
C06754=1112.313,-69.983,-48.239,179.729,5.126,148.964
C06755=1112.308,-69.734,-48.251,179.729,5.131,148.965
C06756=1112.302,-69.484,-48.261,179.729,5.136,148.966
C06757=1112.297,-69.234,-48.273,179.729,5.141,148.967
C06758=1112.292,-68.985,-48.283,179.729,5.146,148.968
C06759=1112.286,-68.735,-48.295,179.730,5.152,148.969
C06760=1112.281,-68.485,-48.305,179.730,5.157,148.970
C06761=1112.276,-68.236,-48.316,179.730,5.162,148.972
C06762=1112.271,-67.986,-48.327,179.730,5.167,148.972
C06763=1112.266,-67.736,-48.339,179.730,5.172,148.974
C06764=1112.260,-67.487,-48.350,179.731,5.178,148.975
C06765=1112.255,-67.236,-48.360,179.731,5.183,148.976
C06766=1112.250,-66.986,-48.372,179.731,5.188,148.977
C06767=1112.245,-66.738,-48.383,179.731,5.193,148.978
C06768=1112.240,-66.487,-48.394,179.731,5.198,148.979
C06769=1112.234,-66.237,-48.405,179.732,5.203,148.980
C06770=1112.229,-65.988,-48.416,179.732,5.209,148.981
C06771=1112.224,-65.739,-48.428,179.732,5.214,148.982
C06772=1112.218,-65.488,-48.439,179.732,5.218,148.983
C06773=1112.213,-65.239,-48.450,179.733,5.223,148.984
C06774=1112.209,-64.990,-48.461,179.733,5.229,148.985
C06775=1112.203,-64.739,-48.472,179.734,5.234,148.986
C06776=1112.197,-64.490,-48.483,179.733,5.239,148.987
C06777=1112.193,-64.241,-48.494,179.734,5.244,148.988
C06778=1112.187,-63.991,-48.506,179.734,5.250,148.989
C06779=1112.182,-63.740,-48.517,179.735,5.254,148.990
C06780=1112.177,-63.491,-48.528,179.735,5.259,148.991
C06781=1112.172,-63.242,-48.540,179.735,5.264,148.992
C06782=1112.167,-62.992,-48.551,179.736,5.270,148.993
C06783=1112.161,-62.743,-48.562,179.736,5.275,148.994
C06784=1112.156,-62.492,-48.573,179.736,5.280,148.995
C06785=1112.150,-62.242,-48.585,179.737,5.285,148.996
C06786=1112.146,-61.993,-48.596,179.738,5.290,148.997
C06787=1112.140,-61.744,-48.607,179.737,5.295,148.998
C06788=1112.135,-61.494,-48.619,179.738,5.300,148.999
C06789=1112.130,-61.244,-48.630,179.738,5.305,149.000
C06790=1112.125,-60.994,-48.641,179.739,5.310,149.001
C06791=1112.120,-60.744,-48.653,179.739,5.315,149.002
C06792=1112.114,-60.495,-48.664,179.739,5.320,149.003
C06793=1112.109,-60.245,-48.676,179.740,5.326,149.004
C06794=1112.104,-59.995,-48.687,179.741,5.331,149.005
C06795=1112.099,-59.781,-48.697,179.741,5.334,149.006
C06796=1112.095,-59.566,-48.707,179.740,5.338,149.007
C06797=1112.090,-59.352,-48.717,179.740,5.342,149.008
C06798=1112.086,-59.137,-48.727,179.740,5.346,149.009
C06799=1112.082,-58.922,-48.737,179.740,5.350,149.010
C06800=1112.078,-58.707,-48.747,179.740,5.355,149.011
C06801=1112.073,-58.493,-48.756,179.740,5.359,149.012
C06802=1112.069,-58.278,-48.766,179.740,5.363,149.012
C06803=1112.063,-58.028,-48.778,179.740,5.367,149.013
C06804=1112.059,-57.779,-48.789,179.740,5.372,149.015
C06805=1112.053,-57.529,-48.801,179.739,5.377,149.016
C06806=1112.048,-57.279,-48.813,179.739,5.381,149.017
C06807=1112.042,-57.030,-48.824,179.739,5.386,149.018
C06808=1112.037,-56.780,-48.836,179.740,5.391,149.019
C06809=1112.032,-56.530,-48.847,179.739,5.395,149.020
C06810=1112.027,-56.280,-48.859,179.739,5.400,149.021
C06811=1112.022,-56.031,-48.870,179.739,5.404,149.022
C06812=1112.017,-55.781,-48.882,179.738,5.409,149.023
C06813=1112.012,-55.531,-48.894,179.738,5.415,149.024
C06814=1112.006,-55.282,-48.905,179.738,5.419,149.025
C06815=1112.001,-55.032,-48.917,179.738,5.424,149.026
C06816=1111.996,-54.782,-48.928,179.739,5.428,149.027
C06817=1111.990,-54.532,-48.940,179.738,5.433,149.028
C06818=1111.986,-54.283,-48.951,179.738,5.438,149.030
C06819=1111.980,-54.033,-48.963,179.738,5.442,149.030
C06820=1111.975,-53.784,-48.976,179.737,5.447,149.032
C06821=1111.970,-53.534,-48.987,179.737,5.452,149.033
C06822=1111.964,-53.285,-48.999,179.737,5.456,149.034
C06823=1111.959,-53.035,-49.011,179.737,5.461,149.035
C06824=1111.954,-52.785,-49.022,179.737,5.466,149.036
C06825=1111.949,-52.535,-49.034,179.737,5.470,149.037
C06826=1111.943,-52.285,-49.046,179.737,5.475,149.038
C06827=1111.939,-52.036,-49.058,179.736,5.480,149.039
C06828=1111.934,-51.786,-49.070,179.737,5.485,149.040
C06829=1111.928,-51.536,-49.081,179.736,5.490,149.041
C06830=1111.924,-51.287,-49.093,179.736,5.494,149.042
C06831=1111.918,-51.037,-49.105,179.736,5.499,149.043
C06832=1111.913,-50.787,-49.117,179.735,5.503,149.045
C06833=1111.908,-50.539,-49.128,179.735,5.508,149.046
C06834=1111.902,-50.289,-49.140,179.735,5.513,149.047
C06835=1111.897,-50.039,-49.152,179.735,5.517,149.048
C06836=1111.891,-49.789,-49.164,179.735,5.522,149.049
C06837=1111.887,-49.540,-49.176,179.735,5.528,149.050
C06838=1111.882,-49.290,-49.188,179.735,5.531,149.051
C06839=1111.876,-49.040,-49.200,179.735,5.537,149.052
C06840=1111.871,-48.790,-49.211,179.734,5.541,149.053
C06841=1111.866,-48.541,-49.223,179.734,5.546,149.054
C06842=1111.861,-48.291,-49.235,179.734,5.551,149.055
C06843=1111.855,-48.041,-49.247,179.734,5.555,149.056
C06844=1111.850,-47.791,-49.259,179.734,5.560,149.058
C06845=1111.846,-47.542,-49.271,179.734,5.565,149.059
C06846=1111.840,-47.292,-49.283,179.733,5.569,149.060
C06847=1111.835,-47.042,-49.295,179.733,5.574,149.061
C06848=1111.830,-46.793,-49.307,179.733,5.578,149.062
C06849=1111.825,-46.543,-49.319,179.733,5.584,149.063
C06850=1111.820,-46.293,-49.331,179.733,5.589,149.064
C06851=1111.816,-46.079,-49.341,179.733,5.593,149.065
C06852=1111.810,-45.864,-49.352,179.733,5.597,149.066
C06853=1111.806,-45.650,-49.362,179.733,5.600,149.067
C06854=1111.801,-45.436,-49.372,179.732,5.604,149.068
C06855=1111.797,-45.221,-49.382,179.732,5.608,149.069
C06856=1111.793,-45.006,-49.392,179.732,5.612,149.070
C06857=1111.788,-44.791,-49.404,179.732,5.616,149.070
C06858=1111.784,-44.576,-49.414,179.732,5.620,149.071
C06859=1111.778,-44.326,-49.426,179.732,5.625,149.073
C06860=1111.773,-44.077,-49.438,179.732,5.630,149.074
C06861=1111.768,-43.828,-49.449,179.731,5.635,149.075
C06862=1111.763,-43.578,-49.462,179.731,5.640,149.076
C06863=1111.758,-43.328,-49.474,179.731,5.645,149.077
C06864=1111.753,-43.079,-49.487,179.731,5.649,149.078
C06865=1111.747,-42.829,-49.498,179.731,5.654,149.079
C06866=1111.742,-42.579,-49.510,179.732,5.659,149.080
C06867=1111.737,-42.330,-49.523,179.732,5.664,149.081
C06868=1111.731,-42.080,-49.535,179.733,5.670,149.082
C06869=1111.727,-41.831,-49.547,179.734,5.675,149.083
C06870=1111.722,-41.580,-49.559,179.735,5.680,149.084
C06871=1111.717,-41.331,-49.572,179.735,5.685,149.084
C06872=1111.712,-41.081,-49.584,179.736,5.689,149.085
C06873=1111.706,-40.832,-49.596,179.737,5.695,149.086
C06874=1111.701,-40.582,-49.608,179.737,5.700,149.087
C06875=1111.696,-40.332,-49.621,179.738,5.705,149.088
C06876=1111.690,-40.082,-49.633,179.739,5.710,149.089
C06877=1111.685,-39.833,-49.645,179.739,5.715,149.090
C06878=1111.680,-39.584,-49.658,179.740,5.719,149.091
C06879=1111.675,-39.334,-49.670,179.741,5.725,149.092
C06880=1111.670,-39.085,-49.682,179.741,5.730,149.093
C06881=1111.665,-38.834,-49.694,179.742,5.734,149.093
C06882=1111.660,-38.585,-49.707,179.743,5.739,149.094
C06883=1111.655,-38.335,-49.720,179.743,5.743,149.095
C06884=1111.649,-38.085,-49.732,179.744,5.748,149.096
C06885=1111.644,-37.836,-49.744,179.744,5.753,149.097
C06886=1111.639,-37.587,-49.757,179.745,5.758,149.098
C06887=1111.633,-37.337,-49.769,179.746,5.763,149.098
C06888=1111.628,-37.087,-49.781,179.746,5.768,149.099
C06889=1111.624,-36.837,-49.794,179.747,5.772,149.100
C06890=1111.618,-36.587,-49.806,179.747,5.777,149.101
C06891=1111.613,-36.338,-49.819,179.748,5.781,149.102
C06892=1111.608,-36.089,-49.831,179.748,5.785,149.103
C06893=1111.603,-35.839,-49.843,179.749,5.790,149.104
C06894=1111.598,-35.589,-49.856,179.749,5.795,149.105
C06895=1111.593,-35.340,-49.869,179.749,5.800,149.105
C06896=1111.587,-35.090,-49.882,179.750,5.804,149.106
C06897=1111.582,-34.840,-49.894,179.751,5.809,149.107
C06898=1111.577,-34.591,-49.906,179.751,5.813,149.108
C06899=1111.572,-34.341,-49.919,179.751,5.817,149.109
C06900=1111.567,-34.091,-49.932,179.752,5.822,149.110
C06901=1111.562,-33.842,-49.945,179.752,5.827,149.111
C06902=1111.556,-33.592,-49.956,179.752,5.832,149.112
C06903=1111.551,-33.343,-49.969,179.753,5.835,149.112
C06904=1111.547,-33.093,-49.982,179.753,5.840,149.113
C06905=1111.541,-32.843,-49.995,179.754,5.845,149.114
C06906=1111.536,-32.594,-50.008,179.754,5.848,149.115
C06907=1111.532,-32.379,-50.018,179.754,5.852,149.116
C06908=1111.527,-32.164,-50.029,179.754,5.857,149.117
C06909=1111.523,-31.950,-50.040,179.755,5.860,149.117
C06910=1111.518,-31.736,-50.051,179.755,5.864,149.118
C06911=1111.514,-31.521,-50.062,179.755,5.868,149.119
C06912=1111.509,-31.307,-50.073,179.755,5.871,149.120
C06913=1111.505,-31.091,-50.084,179.755,5.875,149.120
C06914=1111.501,-30.877,-50.095,179.755,5.879,149.121
C06915=1111.496,-30.627,-50.108,179.756,5.884,149.122
C06916=1111.490,-30.378,-50.120,179.756,5.888,149.123
C06917=1111.485,-30.129,-50.133,179.756,5.893,149.124
C06918=1111.480,-29.878,-50.146,179.756,5.897,149.125
C06919=1111.475,-29.629,-50.159,179.756,5.901,149.126
C06920=1111.470,-29.380,-50.171,179.756,5.905,149.127
C06921=1111.465,-29.130,-50.184,179.756,5.910,149.128
C06922=1111.460,-28.880,-50.197,179.756,5.914,149.129
C06923=1111.454,-28.631,-50.210,179.756,5.918,149.130
C06924=1111.449,-28.382,-50.223,179.756,5.923,149.131
C06925=1111.445,-28.131,-50.236,179.756,5.927,149.132
C06926=1111.439,-27.882,-50.248,179.756,5.932,149.132
C06927=1111.434,-27.633,-50.262,179.756,5.936,149.134
C06928=1111.429,-27.383,-50.275,179.756,5.940,149.134
C06929=1111.424,-27.133,-50.287,179.756,5.945,149.135
C06930=1111.419,-26.884,-50.300,179.756,5.949,149.137
C06931=1111.414,-26.634,-50.313,179.756,5.954,149.137
C06932=1111.408,-26.384,-50.326,179.755,5.958,149.139
C06933=1111.403,-26.135,-50.339,179.755,5.962,149.139
C06934=1111.398,-25.885,-50.352,179.755,5.967,149.141
C06935=1111.393,-25.635,-50.365,179.755,5.971,149.142
C06936=1111.388,-25.386,-50.377,179.756,5.976,149.142
C06937=1111.383,-25.136,-50.390,179.756,5.980,149.143
C06938=1111.377,-24.886,-50.403,179.756,5.986,149.144
C06939=1111.372,-24.637,-50.416,179.757,5.990,149.145
C06940=1111.368,-24.387,-50.429,179.757,5.995,149.146
C06941=1111.362,-24.137,-50.442,179.757,6.000,149.147
C06942=1111.357,-23.888,-50.455,179.758,6.004,149.148
C06943=1111.353,-23.639,-50.469,179.758,6.009,149.149
C06944=1111.347,-23.389,-50.482,179.759,6.014,149.150
C06945=1111.342,-23.139,-50.495,179.759,6.019,149.151
C06946=1111.336,-22.889,-50.508,179.760,6.023,149.152
C06947=1111.331,-22.640,-50.520,179.760,6.028,149.153
C06948=1111.327,-22.390,-50.533,179.761,6.033,149.153
C06949=1111.321,-22.140,-50.547,179.761,6.038,149.154
C06950=1111.316,-21.892,-50.560,179.762,6.042,149.155
C06951=1111.311,-21.641,-50.574,179.762,6.047,149.156
C06952=1111.306,-21.392,-50.586,179.763,6.052,149.157
C06953=1111.301,-21.142,-50.599,179.763,6.057,149.158
C06954=1111.295,-20.892,-50.612,179.764,6.061,149.159
C06955=1111.290,-20.644,-50.626,179.764,6.066,149.160
C06956=1111.285,-20.393,-50.639,179.765,6.071,149.161
C06957=1111.280,-20.144,-50.652,179.765,6.075,149.162
C06958=1111.275,-19.894,-50.665,179.766,6.080,149.162
C06959=1111.270,-19.645,-50.679,179.766,6.084,149.163
C06960=1111.265,-19.395,-50.692,179.766,6.089,149.164
C06961=1111.260,-19.145,-50.705,179.766,6.094,149.165
C06962=1111.255,-18.896,-50.719,179.767,6.098,149.166
C06963=1111.251,-18.681,-50.730,179.768,6.103,149.167
C06964=1111.246,-18.467,-50.741,179.768,6.106,149.167
C06965=1111.241,-18.252,-50.752,179.768,6.110,149.168
C06966=1111.237,-18.038,-50.764,179.769,6.114,149.169
C06967=1111.233,-17.823,-50.776,179.770,6.118,149.170
C06968=1111.228,-17.609,-50.787,179.770,6.123,149.171
C06969=1111.224,-17.394,-50.798,179.770,6.126,149.171
C06970=1111.219,-17.180,-50.810,179.771,6.130,149.172
C06971=1111.215,-16.930,-50.823,179.771,6.135,149.173
C06972=1111.209,-16.681,-50.836,179.772,6.139,149.174
C06973=1111.205,-16.431,-50.850,179.772,6.144,149.175
C06974=1111.199,-16.182,-50.863,179.773,6.149,149.175
C06975=1111.194,-15.932,-50.877,179.773,6.153,149.176
C06976=1111.189,-15.683,-50.890,179.774,6.158,149.177
C06977=1111.183,-15.432,-50.904,179.775,6.162,149.178
C06978=1111.179,-15.184,-50.917,179.775,6.167,149.179
C06979=1111.173,-14.933,-50.931,179.776,6.172,149.180
C06980=1111.168,-14.685,-50.944,179.776,6.176,149.181
C06981=1111.163,-14.434,-50.957,179.777,6.180,149.181
C06982=1111.158,-14.186,-50.971,179.777,6.185,149.182
C06983=1111.153,-13.935,-50.984,179.778,6.190,149.183
C06984=1111.148,-13.686,-50.999,179.778,6.194,149.184
C06985=1111.143,-13.436,-51.011,179.779,6.199,149.185
C06986=1111.138,-13.187,-51.025,179.780,6.203,149.186
C06987=1111.132,-12.937,-51.039,179.780,6.208,149.186
C06988=1111.128,-12.688,-51.052,179.781,6.213,149.187
C06989=1111.122,-12.438,-51.066,179.781,6.218,149.188
C06990=1111.118,-12.188,-51.079,179.781,6.222,149.189
C06991=1111.113,-11.939,-51.094,179.782,6.226,149.190
C06992=1111.107,-11.689,-51.107,179.782,6.231,149.191
C06993=1111.103,-11.440,-51.120,179.783,6.235,149.192
C06994=1111.097,-11.190,-51.134,179.783,6.240,149.192
C06995=1111.092,-10.940,-51.148,179.784,6.244,149.193
C06996=1111.088,-10.690,-51.161,179.785,6.249,149.194
C06997=1111.082,-10.441,-51.175,179.785,6.254,149.195
C06998=1111.077,-10.192,-51.189,179.786,6.259,149.196
C06999=1111.071,-9.942,-51.202,179.787,6.263,149.196
C07000=1111.067,-9.693,-51.216,179.787,6.267,149.197
C07001=1111.062,-9.443,-51.230,179.787,6.272,149.198
C07002=1111.056,-9.193,-51.243,179.788,6.276,149.199
C07003=1111.052,-8.944,-51.257,179.789,6.281,149.200
C07004=1111.047,-8.694,-51.271,179.789,6.285,149.201
C07005=1111.041,-8.445,-51.285,179.790,6.290,149.202
C07006=1111.036,-8.195,-51.299,179.790,6.295,149.203
C07007=1111.031,-7.946,-51.312,179.791,6.299,149.203
C07008=1111.026,-7.696,-51.326,179.792,6.304,149.204
C07009=1111.021,-7.446,-51.340,179.792,6.308,149.205
C07010=1111.016,-7.197,-51.354,179.793,6.312,149.206
C07011=1111.011,-6.947,-51.368,179.793,6.317,149.207
C07012=1111.006,-6.698,-51.382,179.794,6.321,149.207
C07013=1111.001,-6.448,-51.395,179.794,6.326,149.208
C07014=1110.996,-6.199,-51.409,179.795,6.331,149.209
C07015=1110.991,-5.949,-51.424,179.796,6.335,149.210
C07016=1110.985,-5.700,-51.437,179.796,6.340,149.211
C07017=1110.981,-5.450,-51.450,179.797,6.344,149.211
C07018=1110.976,-5.200,-51.465,179.797,6.348,149.212
C07019=1110.971,-4.986,-51.477,179.798,6.353,149.213
C07020=1110.967,-4.772,-51.489,179.798,6.357,149.214
C07021=1110.963,-4.557,-51.500,179.798,6.360,149.215
C07022=1110.957,-4.343,-51.513,179.799,6.364,149.215
C07023=1110.953,-4.128,-51.525,179.800,6.368,149.216
C07024=1110.949,-3.914,-51.538,179.801,6.372,149.217
C07025=1110.945,-3.699,-51.549,179.801,6.376,149.217
C07026=1110.940,-3.485,-51.561,179.801,6.380,149.218
C07027=1110.935,-3.235,-51.576,179.802,6.384,149.219
C07028=1110.930,-2.986,-51.589,179.803,6.389,149.220
C07029=1110.926,-2.737,-51.603,179.803,6.393,149.221
C07030=1110.921,-2.487,-51.617,179.804,6.398,149.221
C07031=1110.916,-2.238,-51.632,179.805,6.403,149.222
C07032=1110.910,-1.989,-51.646,179.805,6.407,149.223
C07033=1110.905,-1.739,-51.660,179.805,6.411,149.224
C07034=1110.900,-1.488,-51.673,179.806,6.415,149.225
C07035=1110.895,-1.239,-51.688,179.807,6.420,149.225
C07036=1110.889,-0.990,-51.702,179.807,6.425,149.226
C07037=1110.884,-0.740,-51.716,179.808,6.429,149.227
C07038=1110.880,-0.490,-51.730,179.809,6.434,149.228
C07039=1110.875,-0.241,-51.744,179.809,6.439,149.229
C07040=1110.870,0.009,-51.759,179.810,6.443,149.230
C07041=1110.864,0.258,-51.773,179.811,6.448,149.230
C07042=1110.859,0.508,-51.787,179.811,6.452,149.231
C07043=1110.854,0.757,-51.802,179.812,6.457,149.232
C07044=1110.849,1.007,-51.816,179.812,6.461,149.233
C07045=1110.845,1.256,-51.830,179.813,6.465,149.234
C07046=1110.839,1.505,-51.844,179.813,6.470,149.235
C07047=1110.834,1.755,-51.859,179.814,6.475,149.235
C07048=1110.829,2.005,-51.873,179.815,6.479,149.236
C07049=1110.824,2.254,-51.887,179.815,6.484,149.237
C07050=1110.819,2.504,-51.901,179.816,6.489,149.238
C07051=1110.814,2.754,-51.916,179.816,6.493,149.239
C07052=1110.809,3.003,-51.930,179.817,6.498,149.239
C07053=1110.804,3.253,-51.944,179.818,6.502,149.240
C07054=1110.799,3.502,-51.959,179.819,6.507,149.241
C07055=1110.794,3.751,-51.973,179.819,6.512,149.242
C07056=1110.789,4.001,-51.987,179.819,6.515,149.243
C07057=1110.784,4.251,-52.002,179.820,6.520,149.244
C07058=1110.778,4.501,-52.017,179.821,6.525,149.245
C07059=1110.773,4.749,-52.031,179.821,6.529,149.245
C07060=1110.768,4.999,-52.046,179.822,6.534,149.246
C07061=1110.763,5.249,-52.060,179.823,6.538,149.247
C07062=1110.758,5.498,-52.074,179.823,6.543,149.248
C07063=1110.753,5.748,-52.088,179.824,6.548,149.249
C07064=1110.749,5.997,-52.103,179.824,6.553,149.250
C07065=1110.744,6.247,-52.118,179.825,6.557,149.250
C07066=1110.738,6.497,-52.133,179.826,6.562,149.251
C07067=1110.733,6.747,-52.147,179.826,6.566,149.252
C07068=1110.729,6.996,-52.162,179.827,6.571,149.253
C07069=1110.723,7.245,-52.176,179.827,6.576,149.254
C07070=1110.718,7.494,-52.190,179.828,6.580,149.255
C07071=1110.713,7.743,-52.205,179.829,6.585,149.255
C07072=1110.708,7.994,-52.220,179.830,6.590,149.256
C07073=1110.703,8.243,-52.234,179.830,6.594,149.257
C07074=1110.698,8.492,-52.249,179.831,6.599,149.258
C07075=1110.694,8.707,-52.261,179.831,6.602,149.259
C07076=1110.689,8.921,-52.274,179.831,6.606,149.259
C07077=1110.685,9.136,-52.287,179.831,6.610,149.260
C07078=1110.681,9.350,-52.299,179.832,6.614,149.261
C07079=1110.676,9.564,-52.312,179.833,6.618,149.262
C07080=1110.672,9.778,-52.324,179.833,6.622,149.262
C07081=1110.668,9.993,-52.337,179.834,6.626,149.263
C07082=1110.663,10.208,-52.350,179.834,6.630,149.264
C07083=1110.659,10.457,-52.365,179.835,6.634,149.265
C07084=1110.654,10.706,-52.379,179.835,6.639,149.266
C07085=1110.648,10.956,-52.394,179.835,6.643,149.266
C07086=1110.643,11.205,-52.408,179.836,6.648,149.267
C07087=1110.638,11.455,-52.423,179.836,6.652,149.268
C07088=1110.633,11.704,-52.438,179.837,6.657,149.269
C07089=1110.628,11.954,-52.453,179.838,6.661,149.270
C07090=1110.623,12.203,-52.468,179.838,6.666,149.271
C07091=1110.618,12.452,-52.482,179.838,6.670,149.272
C07092=1110.613,12.702,-52.497,179.839,6.675,149.272
C07093=1110.608,12.952,-52.512,179.840,6.679,149.273
C07094=1110.604,13.201,-52.527,179.841,6.684,149.274
C07095=1110.598,13.451,-52.542,179.841,6.688,149.275
C07096=1110.593,13.700,-52.557,179.842,6.692,149.276
C07097=1110.588,13.950,-52.571,179.842,6.697,149.276
C07098=1110.583,14.200,-52.587,179.843,6.701,149.277
C07099=1110.578,14.449,-52.601,179.843,6.706,149.278
C07100=1110.573,14.698,-52.616,179.844,6.710,149.279
C07101=1110.568,14.948,-52.632,179.845,6.715,149.280
C07102=1110.563,15.197,-52.646,179.845,6.719,149.281
C07103=1110.558,15.447,-52.661,179.846,6.723,149.281
C07104=1110.553,15.697,-52.676,179.846,6.728,149.282
C07105=1110.548,15.946,-52.691,179.847,6.733,149.283
C07106=1110.543,16.195,-52.706,179.848,6.737,149.284
C07107=1110.538,16.445,-52.721,179.848,6.741,149.285
C07108=1110.533,16.694,-52.736,179.848,6.746,149.285
C07109=1110.528,16.943,-52.751,179.849,6.750,149.286
C07110=1110.523,17.193,-52.766,179.850,6.755,149.287
C07111=1110.518,17.443,-52.781,179.851,6.759,149.288
C07112=1110.513,17.692,-52.796,179.851,6.763,149.289
C07113=1110.508,17.942,-52.811,179.852,6.767,149.289
C07114=1110.503,18.191,-52.826,179.853,6.772,149.290
C07115=1110.497,18.441,-52.842,179.853,6.777,149.291
C07116=1110.493,18.690,-52.856,179.854,6.781,149.292
C07117=1110.488,18.940,-52.871,179.854,6.785,149.292
C07118=1110.483,19.189,-52.887,179.855,6.789,149.293
C07119=1110.478,19.438,-52.902,179.856,6.794,149.294
C07120=1110.473,19.689,-52.917,179.857,6.798,149.295
C07121=1110.468,19.938,-52.932,179.857,6.803,149.296
C07122=1110.463,20.187,-52.948,179.858,6.806,149.296
C07123=1110.458,20.436,-52.963,179.858,6.811,149.297
C07124=1110.452,20.686,-52.977,179.859,6.815,149.298
C07125=1110.447,20.936,-52.993,179.860,6.820,149.299
C07126=1110.443,21.186,-53.008,179.861,6.824,149.299
C07127=1110.438,21.435,-53.024,179.861,6.828,149.300
C07128=1110.433,21.684,-53.039,179.862,6.833,149.301
C07129=1110.428,21.933,-53.055,179.863,6.837,149.302
C07130=1110.423,22.183,-53.069,179.864,6.842,149.302
C07131=1110.418,22.397,-53.083,179.864,6.845,149.303
C07132=1110.415,22.611,-53.096,179.865,6.849,149.304
C07133=1110.410,22.826,-53.108,179.866,6.853,149.304
C07134=1110.405,23.040,-53.122,179.866,6.857,149.305
C07135=1110.402,23.254,-53.135,179.866,6.860,149.306
C07136=1110.397,23.469,-53.148,179.867,6.863,149.306
C07137=1110.392,23.683,-53.161,179.868,6.868,149.307
C07138=1110.389,23.897,-53.175,179.869,6.871,149.307
C07139=1110.383,24.146,-53.190,179.869,6.876,149.308
C07140=1110.378,24.395,-53.206,179.870,6.879,149.309
C07141=1110.374,24.645,-53.221,179.871,6.884,149.310
C07142=1110.368,24.895,-53.237,179.871,6.888,149.310
C07143=1110.364,25.144,-53.252,179.873,6.893,149.311
C07144=1110.358,25.393,-53.267,179.874,6.897,149.312
C07145=1110.354,25.643,-53.283,179.874,6.901,149.313
C07146=1110.349,25.892,-53.298,179.875,6.905,149.313
C07147=1110.344,26.142,-53.314,179.876,6.909,149.314
C07148=1110.338,26.391,-53.329,179.876,6.914,149.315
C07149=1110.334,26.641,-53.345,179.877,6.918,149.316
C07150=1110.329,26.890,-53.360,179.878,6.922,149.316
C07151=1110.323,27.140,-53.376,179.879,6.926,149.317
C07152=1110.318,27.389,-53.392,179.879,6.931,149.318
C07153=1110.314,27.639,-53.407,179.880,6.935,149.318
C07154=1110.309,27.888,-53.422,179.881,6.939,149.319
C07155=1110.303,28.138,-53.438,179.882,6.943,149.320
C07156=1110.298,28.387,-53.453,179.882,6.948,149.321
C07157=1110.294,28.637,-53.469,179.884,6.952,149.321
C07158=1110.288,28.886,-53.485,179.884,6.956,149.322
C07159=1110.283,29.136,-53.500,179.885,6.960,149.323
C07160=1110.279,29.386,-53.516,179.886,6.964,149.323
C07161=1110.274,29.634,-53.532,179.887,6.969,149.324
C07162=1110.268,29.884,-53.547,179.888,6.973,149.325
C07163=1110.264,30.134,-53.563,179.888,6.977,149.325
C07164=1110.259,30.383,-53.578,179.889,6.981,149.326
C07165=1110.254,30.632,-53.594,179.890,6.985,149.327
C07166=1110.249,30.882,-53.610,179.891,6.990,149.327
C07167=1110.244,31.131,-53.626,179.891,6.994,149.328
C07168=1110.238,31.381,-53.642,179.892,6.998,149.329
C07169=1110.234,31.630,-53.657,179.893,7.002,149.330
C07170=1110.229,31.880,-53.673,179.894,7.007,149.330
C07171=1110.224,32.129,-53.688,179.896,7.011,149.331
C07172=1110.219,32.379,-53.705,179.896,7.014,149.332
C07173=1110.214,32.628,-53.721,179.897,7.019,149.332
C07174=1110.209,32.877,-53.736,179.898,7.023,149.333
C07175=1110.204,33.127,-53.752,179.899,7.028,149.334
C07176=1110.199,33.376,-53.768,179.899,7.031,149.334
C07177=1110.194,33.626,-53.784,179.900,7.036,149.335
C07178=1110.189,33.876,-53.799,179.901,7.040,149.336
C07179=1110.184,34.124,-53.816,179.902,7.044,149.336
C07180=1110.179,34.374,-53.832,179.903,7.048,149.337
C07181=1110.174,34.624,-53.847,179.904,7.052,149.338
C07182=1110.169,34.873,-53.864,179.905,7.056,149.338
C07183=1110.165,35.122,-53.879,179.906,7.061,149.339
C07184=1110.159,35.372,-53.894,179.907,7.065,149.340
C07185=1110.155,35.621,-53.911,179.908,7.068,149.340
C07186=1110.149,35.871,-53.927,179.909,7.073,149.341
C07187=1110.145,36.085,-53.940,179.909,7.076,149.342
C07188=1110.141,36.299,-53.954,179.911,7.080,149.342
C07189=1110.136,36.514,-53.968,179.911,7.084,149.343
C07190=1110.132,36.727,-53.982,179.912,7.087,149.343
C07191=1110.128,36.942,-53.996,179.912,7.090,149.344
C07192=1110.123,37.155,-54.009,179.914,7.094,149.344
C07193=1110.119,37.370,-54.023,179.914,7.098,149.345
C07194=1110.115,37.584,-54.037,179.915,7.101,149.345
C07195=1110.110,37.833,-54.053,179.916,7.105,149.346
C07196=1110.105,38.083,-54.069,179.917,7.110,149.347
C07197=1110.100,38.332,-54.086,179.918,7.113,149.347
C07198=1110.095,38.582,-54.101,179.919,7.117,149.348
C07199=1110.090,38.831,-54.118,179.920,7.122,149.349
C07200=1110.085,39.081,-54.134,179.921,7.126,149.349
C07201=1110.080,39.329,-54.150,179.922,7.130,149.350
C07202=1110.075,39.580,-54.166,179.923,7.134,149.350
C07203=1110.070,39.828,-54.182,179.924,7.138,149.351
C07204=1110.065,40.078,-54.198,179.925,7.142,149.352
C07205=1110.060,40.327,-54.214,179.926,7.147,149.352
C07206=1110.055,40.577,-54.230,179.926,7.150,149.353
C07207=1110.050,40.826,-54.247,179.928,7.154,149.354
C07208=1110.046,41.076,-54.263,179.929,7.158,149.354
C07209=1110.041,41.325,-54.279,179.930,7.163,149.355
C07210=1110.036,41.574,-54.296,179.931,7.167,149.356
C07211=1110.031,41.825,-54.311,179.931,7.171,149.356
C07212=1110.026,42.073,-54.328,179.933,7.175,149.357
C07213=1110.021,42.323,-54.345,179.934,7.179,149.357
C07214=1110.016,42.573,-54.361,179.935,7.183,149.358
C07215=1110.011,42.822,-54.377,179.936,7.187,149.359
C07216=1110.006,43.071,-54.393,179.937,7.191,149.359
C07217=1110.001,43.321,-54.410,179.938,7.195,149.360
C07218=1109.996,43.570,-54.426,179.939,7.200,149.361
C07219=1109.992,43.819,-54.443,179.940,7.204,149.361
C07220=1109.986,44.069,-54.458,179.941,7.207,149.362
C07221=1109.981,44.318,-54.475,179.942,7.211,149.362
C07222=1109.977,44.568,-54.492,179.943,7.216,149.363
C07223=1109.971,44.817,-54.508,179.944,7.220,149.364
C07224=1109.967,45.067,-54.524,179.946,7.224,149.364
C07225=1109.962,45.316,-54.541,179.946,7.227,149.365
C07226=1109.957,45.565,-54.557,179.947,7.232,149.365
C07227=1109.952,45.815,-54.574,179.948,7.236,149.366
C07228=1109.947,46.064,-54.590,179.949,7.240,149.367
C07229=1109.942,46.314,-54.607,179.950,7.243,149.367
C07230=1109.937,46.562,-54.623,179.951,7.248,149.368
C07231=1109.933,46.812,-54.640,179.952,7.252,149.368
C07232=1109.927,47.062,-54.656,179.954,7.256,149.369
C07233=1109.922,47.311,-54.673,179.955,7.260,149.369
C07234=1109.917,47.561,-54.689,179.956,7.264,149.370
C07235=1109.913,47.810,-54.706,179.957,7.268,149.371
C07236=1109.907,48.059,-54.723,179.958,7.272,149.371
C07237=1109.903,48.309,-54.740,179.959,7.276,149.372
C07238=1109.898,48.558,-54.756,179.960,7.280,149.372
C07239=1109.893,48.808,-54.772,179.961,7.284,149.373
C07240=1109.888,49.057,-54.789,179.962,7.288,149.374
C07241=1109.883,49.307,-54.806,179.963,7.292,149.374
C07242=1109.878,49.556,-54.822,179.965,7.296,149.375
C07243=1109.873,49.770,-54.837,179.965,7.300,149.375
C07244=1109.869,49.984,-54.851,179.966,7.303,149.376
C07245=1109.865,50.198,-54.865,179.967,7.306,149.376
C07246=1109.862,50.412,-54.880,179.968,7.310,149.377
C07247=1109.857,50.626,-54.894,179.969,7.313,149.377
C07248=1109.853,50.840,-54.909,179.970,7.316,149.378
C07249=1109.849,51.054,-54.923,179.972,7.320,149.378
C07250=1109.844,51.268,-54.937,179.972,7.324,149.379
C07251=1109.839,51.518,-54.954,179.974,7.328,149.379
C07252=1109.834,51.767,-54.970,179.974,7.331,149.380
C07253=1109.830,52.017,-54.987,179.975,7.336,149.381
C07254=1109.825,52.266,-55.005,179.977,7.339,149.381
C07255=1109.820,52.514,-55.021,179.978,7.344,149.382
C07256=1109.814,52.764,-55.039,179.980,7.348,149.382
C07257=1109.810,53.014,-55.055,179.980,7.351,149.383
C07258=1109.805,53.263,-55.072,179.981,7.355,149.383
C07259=1109.800,53.512,-55.089,179.983,7.359,149.384
C07260=1109.795,53.762,-55.106,179.984,7.364,149.384
C07261=1109.790,54.012,-55.123,179.985,7.368,149.385
C07262=1109.785,54.261,-55.139,179.986,7.371,149.386
C07263=1109.780,54.510,-55.156,179.987,7.375,149.386
C07264=1109.775,54.760,-55.173,179.988,7.379,149.387
C07265=1109.771,55.009,-55.190,179.990,7.384,149.387
C07266=1109.766,55.258,-55.208,179.991,7.387,149.388
C07267=1109.761,55.507,-55.224,179.992,7.391,149.388
C07268=1109.755,55.757,-55.241,179.993,7.395,149.389
C07269=1109.751,56.006,-55.258,179.994,7.399,149.389
C07270=1109.746,56.256,-55.275,179.995,7.404,149.390
C07271=1109.741,56.505,-55.293,179.997,7.407,149.391
C07272=1109.736,56.754,-55.309,179.998,7.412,149.391
C07273=1109.731,57.004,-55.326,179.999,7.415,149.392
C07274=1109.726,57.253,-55.343,-180.000,7.419,149.392
C07275=1109.721,57.503,-55.360,-179.998,7.423,149.393
C07276=1109.717,57.752,-55.378,-179.997,7.427,149.393
C07277=1109.712,58.001,-55.394,-179.996,7.431,149.394
C07278=1109.706,58.251,-55.412,-179.995,7.435,149.394
C07279=1109.701,58.500,-55.430,-179.994,7.439,149.395
C07280=1109.697,58.749,-55.446,-179.993,7.443,149.396
C07281=1109.692,58.999,-55.463,-179.991,7.447,149.396
C07282=1109.687,59.249,-55.480,-179.990,7.451,149.397
C07283=1109.682,59.497,-55.498,-179.988,7.455,149.397
C07284=1109.677,59.747,-55.514,-179.988,7.459,149.398
C07285=1109.672,59.996,-55.532,-179.986,7.462,149.398
C07286=1109.667,60.246,-55.550,-179.985,7.467,149.399
C07287=1109.663,60.495,-55.566,-179.984,7.471,149.399
C07288=1109.658,60.744,-55.584,-179.983,7.475,149.400
C07289=1109.653,60.994,-55.601,-179.981,7.479,149.400
C07290=1109.648,61.243,-55.618,-179.980,7.482,149.401
C07291=1109.643,61.493,-55.636,-179.979,7.486,149.401
C07292=1109.638,61.741,-55.653,-179.977,7.490,149.402
C07293=1109.633,61.991,-55.671,-179.976,7.494,149.402
C07294=1109.628,62.240,-55.688,-179.975,7.498,149.403
C07295=1109.624,62.489,-55.705,-179.974,7.503,149.404
C07296=1109.618,62.739,-55.722,-179.973,7.506,149.404
C07297=1109.614,62.988,-55.740,-179.972,7.510,149.405
C07298=1109.609,63.238,-55.757,-179.970,7.514,149.405
C07299=1109.604,63.452,-55.772,-179.969,7.517,149.405
C07300=1109.600,63.665,-55.787,-179.968,7.521,149.406
C07301=1109.596,63.880,-55.802,-179.967,7.524,149.406
C07302=1109.592,64.094,-55.818,-179.966,7.527,149.407
C07303=1109.588,64.307,-55.832,-179.964,7.531,149.407
C07304=1109.583,64.521,-55.847,-179.963,7.534,149.408
C07305=1109.580,64.736,-55.862,-179.963,7.538,149.408
C07306=1109.575,64.950,-55.877,-179.961,7.542,149.409
C07307=1109.570,65.199,-55.895,-179.960,7.545,149.409
C07308=1109.566,65.448,-55.912,-179.959,7.549,149.410
C07309=1109.561,65.698,-55.930,-179.957,7.553,149.410
C07310=1109.556,65.947,-55.948,-179.956,7.557,149.411
C07311=1109.551,66.196,-55.965,-179.955,7.561,149.411
C07312=1109.546,66.445,-55.982,-179.953,7.565,149.412
C07313=1109.541,66.695,-56.000,-179.952,7.569,149.412
C07314=1109.536,66.944,-56.017,-179.951,7.573,149.413
C07315=1109.531,67.193,-56.035,-179.950,7.576,149.413
C07316=1109.526,67.443,-56.053,-179.948,7.580,149.414
C07317=1109.522,67.692,-56.070,-179.947,7.585,149.414
C07318=1109.517,67.941,-56.088,-179.945,7.589,149.415
C07319=1109.512,68.191,-56.106,-179.944,7.593,149.415
C07320=1109.507,68.440,-56.123,-179.943,7.597,149.416
C07321=1109.502,68.689,-56.141,-179.941,7.601,149.416
C07322=1109.497,68.939,-56.159,-179.941,7.604,149.417
C07323=1109.493,69.188,-56.177,-179.939,7.608,149.417
C07324=1109.488,69.437,-56.194,-179.937,7.612,149.418
C07325=1109.483,69.686,-56.212,-179.936,7.616,149.419
C07326=1109.478,69.936,-56.230,-179.935,7.620,149.419
C07327=1109.473,70.185,-56.248,-179.933,7.624,149.419
C07328=1109.468,70.435,-56.265,-179.932,7.628,149.420
C07329=1109.463,70.684,-56.283,-179.931,7.632,149.420
C07330=1109.459,70.934,-56.301,-179.930,7.635,149.421
C07331=1109.454,71.183,-56.319,-179.928,7.640,149.422
C07332=1109.449,71.432,-56.337,-179.927,7.643,149.422
C07333=1109.444,71.682,-56.354,-179.925,7.647,149.422
C07334=1109.439,71.931,-56.372,-179.924,7.652,149.423
C07335=1109.434,72.180,-56.390,-179.923,7.656,149.423
C07336=1109.429,72.429,-56.408,-179.921,7.659,149.424
C07337=1109.425,72.678,-56.426,-179.919,7.663,149.424
C07338=1109.420,72.927,-56.444,-179.918,7.668,149.425
C07339=1109.415,73.177,-56.462,-179.917,7.671,149.425
C07340=1109.410,73.426,-56.480,-179.916,7.675,149.426
C07341=1109.406,73.676,-56.498,-179.915,7.679,149.427
C07342=1109.401,73.925,-56.516,-179.913,7.683,149.427
C07343=1109.396,74.174,-56.534,-179.912,7.687,149.427
C07344=1109.390,74.424,-56.551,-179.910,7.691,149.428
C07345=1109.386,74.673,-56.569,-179.909,7.695,149.428
C07346=1109.381,74.922,-56.587,-179.907,7.699,149.429
C07347=1109.376,75.172,-56.606,-179.906,7.703,149.429
C07348=1109.371,75.421,-56.624,-179.905,7.707,149.430
C07349=1109.367,75.670,-56.642,-179.903,7.711,149.430
C07350=1109.362,75.919,-56.660,-179.901,7.715,149.431
C07351=1109.356,76.168,-56.679,-179.900,7.718,149.431
C07352=1109.351,76.418,-56.697,-179.899,7.722,149.432
C07353=1109.347,76.667,-56.715,-179.898,7.726,149.432
C07354=1109.342,76.917,-56.733,-179.896,7.730,149.433
C07355=1109.337,77.131,-56.748,-179.896,7.734,149.433
C07356=1109.334,77.345,-56.764,-179.895,7.737,149.434
C07357=1109.330,77.558,-56.780,-179.894,7.740,149.434
C07358=1109.326,77.773,-56.795,-179.893,7.743,149.435
C07359=1109.321,77.986,-56.811,-179.892,7.746,149.435
C07360=1109.317,78.199,-56.826,-179.891,7.749,149.436
C07361=1109.313,78.413,-56.843,-179.890,7.753,149.436
